// TIA Portal project "MOVIKIT_POSITIONING_V2.1_e_V15.1_V18" (V18)

(* hardware
DEVICE "S71500/ET200MP-Station_1"  S7-1500 station
   slot 0: "Profilschiene_0"  6ES7 590-1***0-0AA0
   slot 1: "S715xx"  CPU 1516F-3 PN/DP  6ES7 516-3FN00-0AB0  V1.8
DEVICE "SIMATIC 1200-Station_2"  S71200.Device
   slot 0: "S7-1200 Baugruppenträger"  Rack  V1.0
   slot 1: "S712xx"  CPU 1211C AC/DC/Rly  6ES7 211-1BD30-0XB0  V2.0
   slot 101: "CM 1243-5"  CM 1243-5  6GK7 243-5DX30-0XE0  V1.0
DEVICE "SIMATIC 300(1)"  S7-300 station
   slot 0: "Rack 0"  Rail  6ES7 390-1***0-0AA0
   slot 2: "CPU 315F-2 PN/DP"  CPU 315F-2 PN/DP  6ES7 315-2FH13-0AB0  V2.6
      slot 1: "MPI/DP interface_1"  X1
      slot 2: "PROFINET interface_1"  PN-IO
         slot 1: "Port_1"  Port
   slot 4: "DI 8/DO 8x24VDC/0.5A_1"  DI8/DO8 x 24VDC / 0.5A  6ES7 323-1BH01-0AA0
DEVICE "GSD-Geraet_1"  GSD.Device.PN
   slot 0: "Baugruppenträger"  Rack  V1.0
   slot 0: "pos-UDT-s73xx"  MDX90 + CFN21 V4.0
      slot 0: "MDX90 + CFN21 V4.0"  MDX90 + CFN21 V4.0
      slot 1: "PN-IO"  PN-IO
         slot 1: "Port 1 - RJ45 (X40)"  Port 1 - RJ45 (X40)
         slot 2: "Port 2 - RJ45 (X41)"  Port 2 - RJ45 (X41)
   slot 2: "Modul I/O (08 Worte)_1"  Module I/O (08 words)
      slot 0: "Modul I/O (08 Worte)"  Module I/O (08 words)
DEVICE "GSD-Geraet_2"  GSD.Device.PN
   slot 0: "Baugruppenträger"  Rack  V1.0
   slot 0: "pos-UDT-s712xx"  MDX90 + CFN21 V4.0
      slot 0: "MDX90 + CFN21 V4.0"  MDX90 + CFN21 V4.0
      slot 1: "PN-IO"  PN-IO
         slot 1: "Port 1 - RJ45 (X40)"  Port 1 - RJ45 (X40)
         slot 2: "Port 2 - RJ45 (X41)"  Port 2 - RJ45 (X41)
   slot 2: "Modul I/O (08 Worte)_1"  Module I/O (08 words)
      slot 0: "Modul I/O (08 Worte)"  Module I/O (08 words)
   slot 3: "Modul I/O (01 Wort)_1"  Module I/O (01 word)
      slot 0: "Modul I/O (01 Wort)"  Module I/O (01 word)
   slot 4: "Modul I/O (02 Worte)_1"  Module I/O (02 words)
      slot 0: "Modul I/O (02 Worte)"  Module I/O (02 words)
   slot 5: "Modul I/O (04 Worte)_1"  Module I/O (04 words)
      slot 0: "Modul I/O (04 Worte)"  Module I/O (04 words)
DEVICE "GSD-Geraet_4"  GSD.Device.PN
   slot 0: "Baugruppenträger"  Rack  V1.0
   slot 0: "pos-s712xx"  MDX90 + CFN21 V4.0
      slot 0: "MDX90 + CFN21 V4.0"  MDX90 + CFN21 V4.0
      slot 1: "PN-IO"  PN-IO
         slot 1: "Port 1 - RJ45 (X40)"  Port 1 - RJ45 (X40)
         slot 2: "Port 2 - RJ45 (X41)"  Port 2 - RJ45 (X41)
   slot 2: "Modul I/O (08 Worte)_1"  Module I/O (08 words)
      slot 0: "Modul I/O (08 Worte)"  Module I/O (08 words)
DEVICE "GSD-Geraet_3"  GSD.Device.PN
   slot 0: "Baugruppenträger"  Rack  V1.0
   slot 0: "pos-UDT-S715xx"  MDX90 + CFN21 V4.0
      slot 0: "MDX90 + CFN21 V4.0"  MDX90 + CFN21 V4.0
      slot 1: "PN-IO"  PN-IO
         slot 1: "Port 1 - RJ45 (X40)"  Port 1 - RJ45 (X40)
         slot 2: "Port 2 - RJ45 (X41)"  Port 2 - RJ45 (X41)
   slot 2: "Modul I/O (08 Worte)_1"  Module I/O (08 words)
      slot 0: "Modul I/O (08 Worte)"  Module I/O (08 words)
*)

// ===== PLC "S715xx"  CPU 1516F-3 PN/DP =====

VAR_GLOBAL   // PLC tag table "Standard-Variablentabelle"
   "Clock_Byte" AT %MB0 : Byte;
   "Clock_10Hz" AT %M0.0 : Bool;
   "Clock_5Hz" AT %M0.1 : Bool;
   "Clock_2.5Hz" AT %M0.2 : Bool;
   "Clock_2Hz" AT %M0.3 : Bool;
   "Clock_1.25Hz" AT %M0.4 : Bool;
   "Clock_1Hz" AT %M0.5 : Bool;
   "Clock_0.625Hz" AT %M0.6 : Bool;
   "Clock_0.5Hz" AT %M0.7 : Bool;
   "Reset" AT %M1000.0 : Bool;
   "set_ENABLE" AT %M1000.2 : Bool;
   "DRIVES_OFF" AT %M1000.1 : Bool;
   "POS_S715xx_Q" AT %A400.0 : "SEW_MOVIKIT_PositioningDrive_SETPOINTS_V2.1";   // Dieses UDT bildet die 5 Prozeßausgangsdaten der Funktion "Parameterkanal über Prozeßdaten" ab. This UDT maps the 5 process output data of the function "parameter channel via process data".
   "POS_S715xx_I" AT %E400.0 : "SEW_MOVIKIT_PositioningDrive_STATUS_V2.1";   // Dieses UDT bildet die 5 Prozeßeingangsdaten der Funktion "Parameterkanal über Prozeßdaten" ab. This UDT maps the 5 process input data of the function "parameter channel via process data"..
   "pos-plus-S715xx _Start" AT %M1001.7 : Bool;
   "Status (FCB)" AT %MW1004 : Int;
   "SubFault_Fault" AT %MW1024 : Word;
   "Fault" AT %MB1024 : SInt;
   "SubFault" AT %MB1025 : SInt;
   "pos-UDT-S715xx_PO1" AT %AW400 : Word;   // control word
   "pos-UDT-S715xx_PO2" AT %QW402 : Int;   // setpoint speed
   "pos-UDT-S715xx_PO3" AT %QW404 : Int;   // acceleration
   "pos-UDT-S715xx_PO4" AT %QW406 : Int;   // deceleration
   "pos-UDT-S715xx_PO5" AT %QW408 : Word;   // dig. Outputs
   "pos-UDT-S715xx_PI1" AT %IW400 : Int;   // status word
   "pos-UDT-S715xx_PI2" AT %IW402 : Int;   // actual speed
   "pos-UDT-S715xx_PI3" AT %IW404 : Word;   // Status/Main/Subfault
   "pos-UDT-S715xx_PI4" AT %IW406 : Int;   // actual torque
   "pos-UDT-S715xx_PI5" AT %IW408 : Word;   // dig. Inputs
   "pos-UDT-S715xx_PO6" AT %QW410 : Int;   // Target application mode
   "pos-UDT-S715xx_PO7-8" AT %QD412 : DInt;   // Target position
   "pos-UDT-S715xx_PI6" AT %IW416 : Int;   // actual application mode
   "pos-UDT-S715xx_PI7-8" AT %ID418 : DInt;   // actual position
END_VAR

TYPE "SEW_MOVIKIT_PositioningDrive_SETPOINTS_V2.1"
TITLE = SEW_MOVIKIT_PositioningDrive_SETPOINTS
// Dieses UDT bildet die 8 Prozeßeingangsdaten des MOVIKIT PositioningDrives ab. This UDT maps the 8 process input data of the MOVIKIT PositioningDrive.
   STRUCT
      x_Bit_8_Fault_Reset : Bool;
      x_Bit_9_Reserved : Bool;
      x_Bit_10_Activate_DriveTrain2 : Bool;
      x_Bit_11_Reserved : Bool;
      x_Bit_12_Deactivate_SW_Limit_switches : Bool;
      x_Bit_13_Activate_Output_Stage_Inhibit : Bool;
      x_Bit_14_Activate_StandBy_Mode : Bool;
      x_Bit_15_Heartbeat_IN : Bool;
      x_Bit_0_Enable_Emergency_Stop : Bool;
      x_Bit_1_Enable_Application_Stop : Bool;
      x_Bit_2_Reserved : Bool;
      x_Bit_3_Release_Brake : Bool;
      x_Bit_4_Jog_positive : Bool;
      x_Bit_5_Jog_negative : Bool;
      x_Bit_6_Apply_relative_Position : Bool;
      x_Bit_7_Start_Stop : Bool;
      iSetpoint_Speed : Int;
      iSetpoint_Acceleration : Int;
      iSetpoint_Deceleration : Int;
      wDigital_Outputs : Word;
      iSetpointApplicationMode : Int;
      diTargetPosition : DInt;
   END_STRUCT;
END_TYPE

TYPE "SEW_MOVIKIT_PositioningDrive_STATUS_V2.1"
TITLE = SEW_MOVIKIT_PositioningDrive_STATUS
// Dieses UDT bildet die 8 Prozeßausgangsdaten des MOVIKIT PositioningDrives ab. This UDT maps the 8 process output data of the MOVIKIT PositioningDrive.
   STRUCT
      x_Bit_8_Fault : Bool;
      x_Bit_9_Warning : Bool;
      x_Bit_10_DriveTrain2_active : Bool;
      x_Bit_11_Setp_actual_speed_comp_signal_active : Bool;
      x_Bit_12_SW_Limit_switches_inactive : Bool;
      x_Bit_13_Reserved : Bool;
      x_Bit_14_StandBy_mode_active : Bool;
      x_Bit_15_Heartbeat_OUT : Bool;
      x_Bit_0_Ready : Bool;
      x_Bit_1_STO_inactive : Bool;
      x_Bit_2_Output_Stage_enabled : Bool;
      x_Bit_3_Brake_released : Bool;
      x_Bit_4_Motor_turning : Bool;
      x_Bit_5_Active_Drive_referenced : Bool;
      x_Bit_6_New_Relative_Position_applied : Bool;
      x_Bit_7_In_Position_signal_active : Bool;
      iActual_Speed : Int;
      wStatus_main_fault_sub_fault : Word;
      iActual_Torque : Int;
      wDigital_Inputs : Word;
      iActual_Application_Mode : Int;
      diActual_Position : DInt;
   END_STRUCT;
END_TYPE

TYPE "SEW_MOVIKIT_5_PD_PAR_STATUS_V2.0"
   STRUCT
      x_Bit_8_READ_Service_selected : Bool;
      x_Bit_9_WRITE_Service_selected : Bool;
      x_Bit_10 : Bool;
      x_Bit_11 : Bool;
      x_Bit_12 : Bool;
      x_Bit_13_Service_active : Bool;
      x_Bit_14_Service_completed : Bool;
      x_Bit_15_Service_failed : Bool;
      x_Bit_0 : Bool;
      x_Bit_1 : Bool;
      x_Bit_2 : Bool;
      x_Bit_3 : Bool;
      x_Bit_4 : Bool;
      x_Bit_5 : Bool;
      x_Bit_6 : Bool;
      x_Bit_7 : Bool;
      i_actual_Index : Int;
      b_actual_SubIndex : Byte;
      b_actual_Offset : Byte;
      dw_value_read : DWord;
   END_STRUCT;
END_TYPE

TYPE "SEW_MOVIKIT_Function_torque_limit_STATUS_V2.0"
   STRUCT
      x_Bit_8 : Bool;
      x_Bit_9 : Bool;
      x_Bit_10 : Bool;
      x_Bit_11 : Bool;
      x_Bit_12 : Bool;
      x_Bit_13 : Bool;
      x_Bit_14 : Bool;
      x_Bit_15 : Bool;
      x_Bit_0_torque_limit_via_PD_active : Bool;
      x_Bit_1_speed_and_lag_error_monitoring_inactive : Bool;
      x_Bit_2_torque_limit_reached : Bool;
      x_Bit_3_speed_monitoring_inactive : Bool;
      x_Bit_4 : Bool;
      x_Bit_5 : Bool;
      x_Bit_6 : Bool;
      x_Bit_7 : Bool;
      i_actual_torque : Int;
   END_STRUCT;
END_TYPE

TYPE "SEW_MOVIKIT_5_PD_PAR_SETPOINTS_V2.0"
   STRUCT
      x_Bit_8_READ : Bool;
      x_Bit_9_WRITE : Bool;
      x_Bit_10 : Bool;
      x_Bit_11 : Bool;
      x_Bit_12 : Bool;
      x_Bit_13 : Bool;
      x_Bit_14_execute_function : Bool;
      x_Bit_15 : Bool;
      x_Bit_0 : Bool;
      x_Bit_1 : Bool;
      x_Bit_2 : Bool;
      x_Bit_3 : Bool;
      x_Bit_4 : Bool;
      x_Bit_5 : Bool;
      x_Bit_6 : Bool;
      x_Bit_7 : Bool;
      i_Index : Int;
      b_SubIndex : Byte;
      b_Offset : Byte;
      dw_value : DWord;
   END_STRUCT;
END_TYPE

TYPE "SEW_MOVIKIT_Function_torque_limit_SETPOINTS_V2.0"
   STRUCT
      x_Bit_8 : Bool;
      x_Bit_9 : Bool;
      x_Bit_10 : Bool;
      x_Bit_11 : Bool;
      x_Bit_12 : Bool;
      x_Bit_13 : Bool;
      x_Bit_14 : Bool;
      x_Bit_15 : Bool;
      x_Bit_0_activate_torque_limit_via_PD : Bool;
      x_Bit_1_deactivate_monitoring_of_speed_and_lag_error : Bool;
      x_Bit_2 : Bool;
      x_Bit_3_deactivate_speed_monitoring : Bool;
      x_Bit_4 : Bool;
      x_Bit_5 : Bool;
      x_Bit_6 : Bool;
      x_Bit_7 : Bool;
      i_maximum_torque : Int;
   END_STRUCT;
END_TYPE

TYPE "SEW_MOVIKIT_Function_touchprobe_STATUS_V2.0"
   STRUCT
      x_Bit_8 : Bool;
      x_Bit_9 : Bool;
      x_Bit_10 : Bool;
      x_Bit_11 : Bool;
      x_Bit_12 : Bool;
      x_Bit_13 : Bool;
      x_Bit_14 : Bool;
      x_Bit_15 : Bool;
      x_Bit_0_wait_for_trigger : Bool;
      x_Bit_1_trigger_activated : Bool;
      x_Bit_2_maximum_position_reached : Bool;
      x_Bit_3_touchprobe_travel_aborted : Bool;
      x_Bit_4 : Bool;
      x_Bit_5 : Bool;
      x_Bit_6 : Bool;
      x_Bit_7 : Bool;
      "i_counter_touchprobe 1" : Int;
      "di_detected_value_touchprobe 1" : DInt;
   END_STRUCT;
END_TYPE

TYPE "SEW_MOVIKIT_Function_touchprobe_SETPOINTS_V2.0"
   STRUCT
      x_Bit_8 : Bool;
      x_Bit_9 : Bool;
      x_Bit_10 : Bool;
      x_Bit_11 : Bool;
      x_Bit_12 : Bool;
      x_Bit_13 : Bool;
      x_Bit_14 : Bool;
      x_Bit_15 : Bool;
      x_Bit_0_activate_touchprobe_1 : Bool;
      x_Bit_1_activate_length_measurement : Bool;
      x_Bit_2 : Bool;
      x_Bit_3 : Bool;
      x_Bit_4 : Bool;
      x_Bit_5 : Bool;
      x_Bit_6 : Bool;
      x_Bit_7 : Bool;
      i_debouncing_time_for_length_measurement : Int;
      di_relative_position : DInt;
   END_STRUCT;
END_TYPE

FUNCTION "UDT_Positioning_Drive_example" : Void   // FC98, FBD
TITLE = Call the drive "pos-UDT-S715xx"
{ S7_Optimized_Access := 'TRUE' }
AUTHOR : SVSPASE
FAMILY : MOVIKIT
VERSION : 2.0
// This sample program only demonstrates the basic approach. We do not accept any legal or other liability for incorrect program functions and their consequences!
// 
// Please take note of the manual "MOVIKIT® Positioning, Velocity"
// 
// The UDTs "SEW_MOVIKIT_PositioningDrive_SETPOINTS_V2.1" and "SEW_MOVIKIT_PositioningDrive_STATUS_V2.1" are needed. Please make sure that the PLC data types are available in your TIA project.  These UDTs can be copied from the original TIA sample project or from the MOVIKIT_Vel_&_Pos_UDTs_V2.1.al14 library.
// 
// The plc tag "VELOCITY_S715xx_Q" has been assigned to the data type "SEW_MOVIKIT_PositioningDrive_SETPOINTS_V2.1" and  address Q400.0
// 
// The plc tag "VELOCITY_S715xx_I" has been assigned to the data type "SEW_MOVIKIT_PositioningDrive_STATUS_V2.1" and  address I400.0
BEGIN

REGION Network 1: Mapping of Status/Main fault/Subfault
   // If there is no fault or warning, the current FCB is output in "Status (FCB) MW1004 ).
   // 
   // If there is a fault or warning, the Subfault is copied in MB1024 and the Main fault in MB1025
   // 
   // => See "watch table "pos-UDT-S715xx"
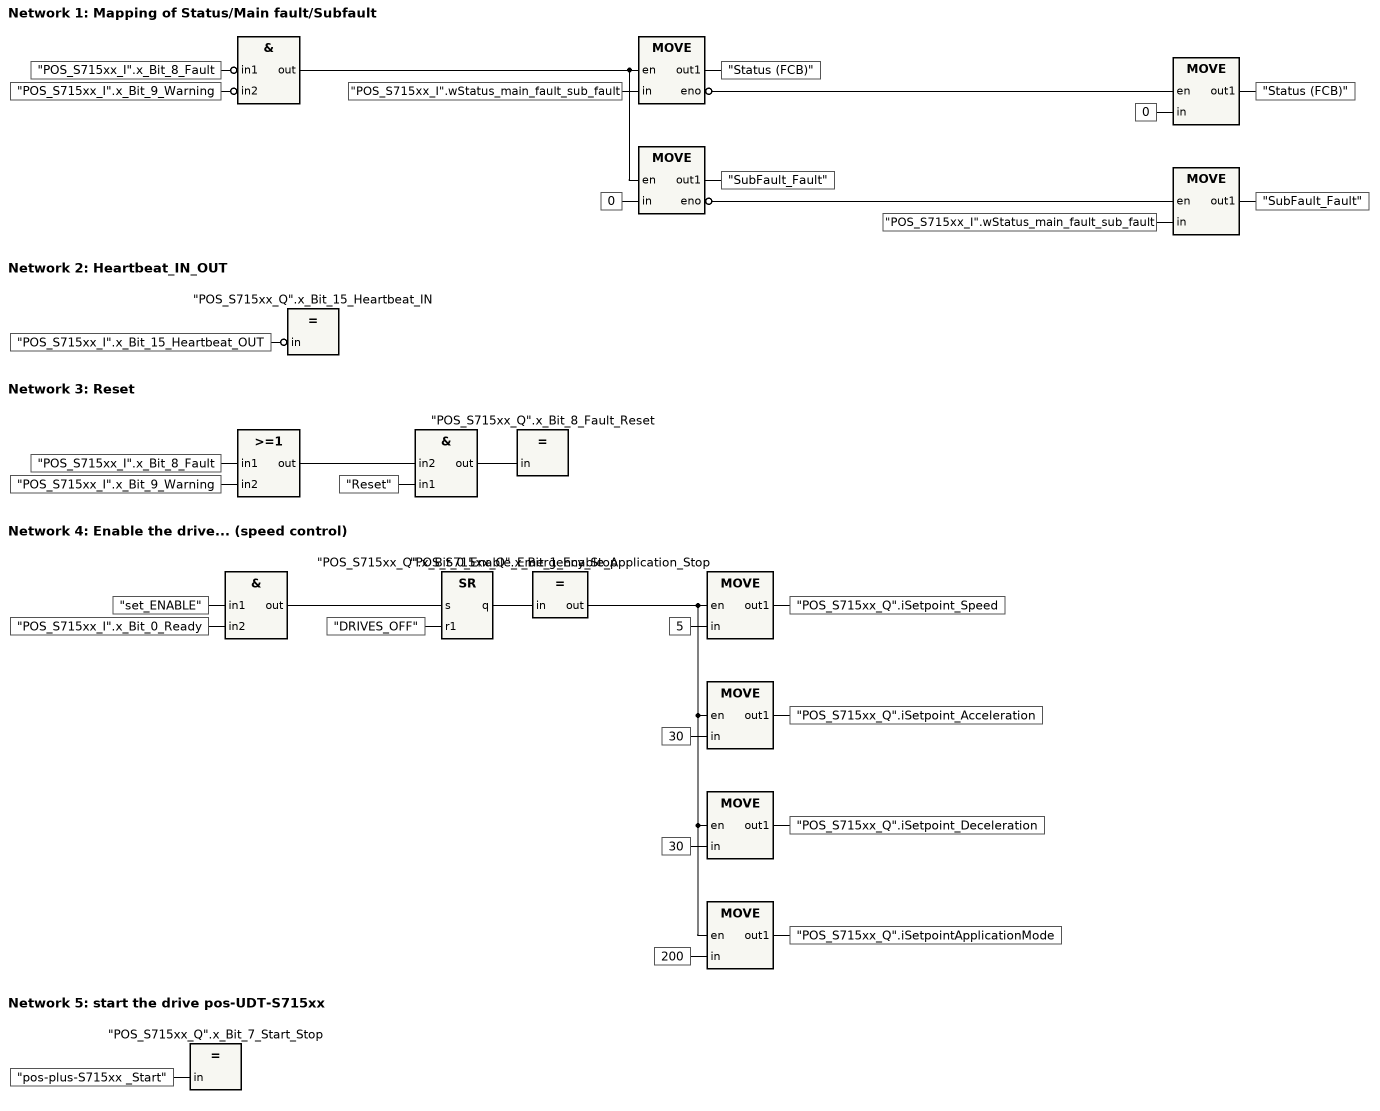
   IF NOT "POS_S715xx_I".x_Bit_8_Fault AND NOT "POS_S715xx_I".x_Bit_9_Warning THEN
       "Status (FCB)" := "POS_S715xx_I".wStatus_main_fault_sub_fault;
   END_IF;
   IF NOT (NOT "POS_S715xx_I".x_Bit_8_Fault AND NOT "POS_S715xx_I".x_Bit_9_Warning) THEN
       "Status (FCB)" := 0;
   END_IF;
   IF NOT "POS_S715xx_I".x_Bit_8_Fault AND NOT "POS_S715xx_I".x_Bit_9_Warning THEN
       "SubFault_Fault" := 0;
   END_IF;
   IF NOT (NOT "POS_S715xx_I".x_Bit_8_Fault AND NOT "POS_S715xx_I".x_Bit_9_Warning) THEN
       "SubFault_Fault" := "POS_S715xx_I".wStatus_main_fault_sub_fault;
   END_IF;
END_REGION

REGION Network 2: Heartbeat_IN_OUT
   "POS_S715xx_Q".x_Bit_15_Heartbeat_IN := NOT "POS_S715xx_I".x_Bit_15_Heartbeat_OUT;
END_REGION

REGION Network 3: Reset
   "POS_S715xx_Q".x_Bit_8_Fault_Reset := ("POS_S715xx_I".x_Bit_8_Fault OR "POS_S715xx_I".x_Bit_9_Warning) AND "Reset";
END_REGION

REGION Network 4: Enable the drive... (speed control)
   // - set enable
   // - assign setpoint speed, acceleration,..,.....
   IF "set_ENABLE" AND "POS_S715xx_I".x_Bit_0_Ready THEN
       "POS_S715xx_Q".x_Bit_0_Enable_Emergency_Stop := TRUE;   // SR flip-flop
   END_IF;
   IF "DRIVES_OFF" THEN "POS_S715xx_Q".x_Bit_0_Enable_Emergency_Stop := FALSE; END_IF;
   "POS_S715xx_Q".x_Bit_1_Enable_Application_Stop := "POS_S715xx_Q".x_Bit_0_Enable_Emergency_Stop;
   IF "POS_S715xx_Q".x_Bit_0_Enable_Emergency_Stop THEN
       "POS_S715xx_Q".iSetpoint_Speed := 5;
       "POS_S715xx_Q".iSetpoint_Acceleration := 30;
       "POS_S715xx_Q".iSetpoint_Deceleration := 30;
       "POS_S715xx_Q".iSetpointApplicationMode := 200;
   END_IF;
END_REGION

REGION Network 5: start the drive pos-UDT-S715xx
   "POS_S715xx_Q".x_Bit_7_Start_Stop := "pos-plus-S715xx _Start";
END_REGION
END_FUNCTION

ORGANIZATION_BLOCK "Main"   // OB1, STL, ProgramCycle
TITLE = "Main Program Sweep (Cycle)"
{ S7_Optimized_Access := 'FALSE' }
VERSION : 0.1
// This sample program only demonstrates the basic approach. We do not accept any legal or other liability for incorrect program functions and their consequences!
// 
// Please take note of the manual "MOVIKIT® Positioning, Velocity"
   VAR_TEMP
      OB1_EV_CLASS : Byte;   // Bits 0-3 = 1 (Coming event), Bits 4-7 = 1 (Event class 1)
      OB1_SCAN_1 : Byte;   // 1 (Cold restart scan 1 of OB 1), 3 (Scan 2-n of OB 1)
      OB1_PRIORITY : Byte;   // Priority of OB Execution
      OB1_OB_NUMBR : Byte;   // 1 (Organization block 1, OB1)
      OB1_RESERVED_1 : Byte;   // Reserved for system
      OB1_RESERVED_2 : Byte;   // Reserved for system
      OB1_PREV_CYCLE : Int;   // Cycle time of previous OB1 scan (milliseconds)
      OB1_MIN_CYCLE : Int;   // Minimum cycle time of OB1 (milliseconds)
      OB1_MAX_CYCLE : Int;   // Maximum cycle time of OB1 (milliseconds)
      OB1_DATE_TIME : Date_And_Time;   // Date and time OB1 started
   END_VAR
BEGIN

REGION Network 1: Call the drive "velocity-UDT-S715xx"

         CALL  "UDT_Positioning_Drive_example";
END_REGION
END_ORGANIZATION_BLOCK

// ===== PLC "S712xx"  CPU 1211C AC/DC/Rly =====

VAR_GLOBAL   // PLC tag table "Standard-Variablentabelle"
   "Clock_Byte" AT %MB0 : Byte;
   "Clock_10Hz" AT %M0.0 : Bool;
   "Clock_5Hz" AT %M0.1 : Bool;
   "Clock_2.5Hz" AT %M0.2 : Bool;
   "Clock_2Hz" AT %M0.3 : Bool;
   "Clock_1.25Hz" AT %M0.4 : Bool;
   "Clock_1Hz" AT %M0.5 : Bool;
   "Clock_0.625Hz" AT %M0.6 : Bool;
   "Clock_0.5Hz" AT %M0.7 : Bool;
   "pos-UDT-S712xx_PO9_Jerk_Time" AT %QW316 : Int;   // Slot 3: jerk time
   "pos-S712xx_PO1" AT %QW330 : Int;   // control word
   "pos-S712xx_PO2" AT %QW332 : Int;   // setpoint speed
   "pos-S712xx_PO3" AT %QW334 : Int;   // acceleration
   "pos-S712xx_PO4" AT %QW336 : Int;   // deceleration
   "pos-S712xx_PO5" AT %QW338 : Int;   // dig. Outputs
   "pos-S712xx_PI1" AT %IW330 : Int;   // status word
   "pos-S712xx_PI2" AT %IW332 : Int;   // actual speed
   "pos-S712xx_PI3" AT %IW334 : Int;   // Status/Main/Subfault
   "pos-S712xx_PI4" AT %IW336 : Int;   // actual torque
   "pos-S712xx_PI5" AT %IW338 : Int;   // dig. Inputs
   "pos-UDT-S712xx_PO1" AT %QW300 : Int;   // Slot 2: control word
   "pos-UDT-S712xx_PO2" AT %QW302 : Int;   // Slot 2: setpoint speed
   "pos-UDT-S712xx_PO3" AT %QW304 : Int;   // Slot 2: acceleration
   "pos-UDT-S712xx_PO4" AT %QW306 : Int;   // Slot 2: deceleration
   "pos-UDT-S712xx_PO5" AT %QW308 : Word;   // Slot 2: dig. Outputs
   "pos-UDT-S712xx_PI1" AT %IW300 : Word;   // Slot 2: status word
   "pos-UDT-S712xx_PI2" AT %IW302 : Int;   // Slot 2: actual speed
   "pos-UDT-S712xx_PI3" AT %IW304 : Int;   // Slot 2: Status/Main/Subfault
   "pos-UDT-S712xx_PI4" AT %IW306 : Int;   // Slot 2: actual torque
   "pos-UDT-S712xx_PI5" AT %IW308 : Int;   // Slot 2: dig. Inputs
   "pos-UDT-S712xx_PI6" AT %IW310 : Int;   // Slot 2: actual application mode
   "pos-UDT-S712xx_PI7-8" AT %ID312 : DInt;   // Slot 2: actual position
   "pos-UDT-S712xx_PI9" AT %IW316 : Int;   // Slot 3: reserved
   "pos-UDT-S712xx_PI10" AT %IW318 : Int;   // Slot 4: Status word for torque limit
   "pos-UDT-S712xx_PI11" AT %IW320 : Int;   // Slot 4: Acual torque
   "pos-UDT-S712xx_PI12" AT %IW322 : Word;   // Slot 5: Status word for positioning via touchprobe
   "pos-S712xx_PO6" AT %QW340 : Int;   // target application mode
   "pos-S712xx_PO7-8" AT %QD342 : DInt;   // target position
   "pos-S712xx_PI6" AT %IW340 : Int;   // actual application mode
   "pos-S712xx_PI7-8" AT %ID342 : DInt;   // actual position
   "pos-UDT-S712xx_PO6" AT %QW310 : Int;   // Slot 2: target application mode
   "pos-UDT-S712xx_PO7-8" AT %QD312 : DInt;   // Slot 2: Target position
   "pos-UDT-S712xx_PO10" AT %QW318 : Word;   // Slot 4: Control word for torque limit
   "pos-UDT-S712xx_PO11" AT %QW320 : Int;   // Slot 4: Maximum Torque
   "pos-UDT-S712xx_PO12" AT %QW322 : Word;   // Slot 5: Control word for pos. via touch probe
   "pos-UDT-S712xx_PO13" AT %QW324 : Int;   // Slot 5: Debouncing time for length measurement
   "pos-UDT-S712xx_PO14-15" AT %QD326 : DInt;   // Slot 5: relative position
   "pos-UDT-S712xx_PI13" AT %IW324 : Int;   // Slot 5: Counter Touch probe 1
   "pos-UDT-S712xx_PI4-15" AT %ID326 : DInt;   // Slot 5: detected value touchprobe 1
END_VAR

TYPE "SEW_MOVIKIT_PositioningDrive_SETPOINTS_V2.1"
TITLE = SEW_MOVIKIT_PositioningDrive_SETPOINTS
// Dieses UDT bildet die 8 Prozeßeingangsdaten des MOVIKIT PositioningDrives ab. This UDT maps the 8 process input data of the MOVIKIT PositioningDrive.
   STRUCT
      x_Bit_8_Fault_Reset : Bool;
      x_Bit_9_Reserved : Bool;
      x_Bit_10_Activate_DriveTrain2 : Bool;
      x_Bit_11_Reserved : Bool;
      x_Bit_12_Deactivate_SW_Limit_switches : Bool;
      x_Bit_13_Activate_Output_Stage_Inhibit : Bool;
      x_Bit_14_Activate_StandBy_Mode : Bool;
      x_Bit_15_Heartbeat_IN : Bool;
      x_Bit_0_Enable_Emergency_Stop : Bool;
      x_Bit_1_Enable_Application_Stop : Bool;
      x_Bit_2_Reserved : Bool;
      x_Bit_3_Release_Brake : Bool;
      x_Bit_4_Jog_positive : Bool;
      x_Bit_5_Jog_negative : Bool;
      x_Bit_6_Apply_relative_Position : Bool;
      x_Bit_7_Start_Stop : Bool;
      iSetpoint_Speed : Int;
      iSetpoint_Acceleration : Int;
      iSetpoint_Deceleration : Int;
      wDigital_Outputs : Word;
      iSetpointApplicationMode : Int;
      diTargetPosition : DInt;
   END_STRUCT;
END_TYPE

TYPE "SEW_MOVIKIT_PositioningDrive_STATUS_V2.1"
TITLE = SEW_MOVIKIT_PositioningDrive_STATUS
// Dieses UDT bildet die 8 Prozeßausgangsdaten des MOVIKIT PositioningDrives ab. This UDT maps the 8 process output data of the MOVIKIT PositioningDrive.
   STRUCT
      x_Bit_8_Fault : Bool;
      x_Bit_9_Warning : Bool;
      x_Bit_10_DriveTrain2_active : Bool;
      x_Bit_11_Setp_actual_speed_comp_signal_active : Bool;
      x_Bit_12_SW_Limit_switches_inactive : Bool;
      x_Bit_13_Reserved : Bool;
      x_Bit_14_StandBy_mode_active : Bool;
      x_Bit_15_Heartbeat_OUT : Bool;
      x_Bit_0_Ready : Bool;
      x_Bit_1_STO_inactive : Bool;
      x_Bit_2_Output_Stage_enabled : Bool;
      x_Bit_3_Brake_released : Bool;
      x_Bit_4_Motor_turning : Bool;
      x_Bit_5_Active_Drive_referenced : Bool;
      x_Bit_6_New_Relative_Position_applied : Bool;
      x_Bit_7_In_Position_signal_active : Bool;
      iActual_Speed : Int;
      wStatus_main_fault_sub_fault : Word;
      iActual_Torque : Int;
      wDigital_Inputs : Word;
      iActual_Application_Mode : Int;
      diActual_Position : DInt;
   END_STRUCT;
END_TYPE

TYPE "SEW_MOVIKIT_5_PD_PAR_STATUS_V2.0"
   STRUCT
      x_Bit_8_READ_Service_selected : Bool;
      x_Bit_9_WRITE_Service_selected : Bool;
      x_Bit_10 : Bool;
      x_Bit_11 : Bool;
      x_Bit_12 : Bool;
      x_Bit_13_Service_active : Bool;
      x_Bit_14_Service_completed : Bool;
      x_Bit_15_Service_failed : Bool;
      x_Bit_0 : Bool;
      x_Bit_1 : Bool;
      x_Bit_2 : Bool;
      x_Bit_3 : Bool;
      x_Bit_4 : Bool;
      x_Bit_5 : Bool;
      x_Bit_6 : Bool;
      x_Bit_7 : Bool;
      i_actual_Index : Int;
      b_actual_SubIndex : Byte;
      b_actual_Offset : Byte;
      dw_value_read : DWord;
   END_STRUCT;
END_TYPE

TYPE "SEW_MOVIKIT_Function_torque_limit_STATUS_V2.0"
   STRUCT
      x_Bit_8 : Bool;
      x_Bit_9 : Bool;
      x_Bit_10 : Bool;
      x_Bit_11 : Bool;
      x_Bit_12 : Bool;
      x_Bit_13 : Bool;
      x_Bit_14 : Bool;
      x_Bit_15 : Bool;
      x_Bit_0_torque_limit_via_PD_active : Bool;
      x_Bit_1_speed_and_lag_error_monitoring_inactive : Bool;
      x_Bit_2_torque_limit_reached : Bool;
      x_Bit_3_speed_monitoring_inactive : Bool;
      x_Bit_4 : Bool;
      x_Bit_5 : Bool;
      x_Bit_6 : Bool;
      x_Bit_7 : Bool;
      i_actual_torque : Int;
   END_STRUCT;
END_TYPE

TYPE "SEW_MOVIKIT_5_PD_PAR_SETPOINTS_V2.0"
   STRUCT
      x_Bit_8_READ : Bool;
      x_Bit_9_WRITE : Bool;
      x_Bit_10 : Bool;
      x_Bit_11 : Bool;
      x_Bit_12 : Bool;
      x_Bit_13 : Bool;
      x_Bit_14_execute_function : Bool;
      x_Bit_15 : Bool;
      x_Bit_0 : Bool;
      x_Bit_1 : Bool;
      x_Bit_2 : Bool;
      x_Bit_3 : Bool;
      x_Bit_4 : Bool;
      x_Bit_5 : Bool;
      x_Bit_6 : Bool;
      x_Bit_7 : Bool;
      i_Index : Int;
      b_SubIndex : Byte;
      b_Offset : Byte;
      dw_value : DWord;
   END_STRUCT;
END_TYPE

TYPE "SEW_MOVIKIT_Function_torque_limit_SETPOINTS_V2.0"
   STRUCT
      x_Bit_8 : Bool;
      x_Bit_9 : Bool;
      x_Bit_10 : Bool;
      x_Bit_11 : Bool;
      x_Bit_12 : Bool;
      x_Bit_13 : Bool;
      x_Bit_14 : Bool;
      x_Bit_15 : Bool;
      x_Bit_0_activate_torque_limit_via_PD : Bool;
      x_Bit_1_deactivate_monitoring_of_speed_and_lag_error : Bool;
      x_Bit_2 : Bool;
      x_Bit_3_deactivate_speed_monitoring : Bool;
      x_Bit_4 : Bool;
      x_Bit_5 : Bool;
      x_Bit_6 : Bool;
      x_Bit_7 : Bool;
      i_maximum_torque : Int;
   END_STRUCT;
END_TYPE

TYPE "SEW_MOVIKIT_Function_touchprobe_STATUS_V2.0"
   STRUCT
      x_Bit_8 : Bool;
      x_Bit_9 : Bool;
      x_Bit_10 : Bool;
      x_Bit_11 : Bool;
      x_Bit_12 : Bool;
      x_Bit_13 : Bool;
      x_Bit_14 : Bool;
      x_Bit_15 : Bool;
      x_Bit_0_wait_for_trigger : Bool;
      x_Bit_1_trigger_activated : Bool;
      x_Bit_2_maximum_position_reached : Bool;
      x_Bit_3_touchprobe_travel_aborted : Bool;
      x_Bit_4 : Bool;
      x_Bit_5 : Bool;
      x_Bit_6 : Bool;
      x_Bit_7 : Bool;
      "i_counter_touchprobe 1" : Int;
      "di_detected_value_touchprobe 1" : DInt;
   END_STRUCT;
END_TYPE

TYPE "SEW_MOVIKIT_Function_touchprobe_SETPOINTS_V2.0"
   STRUCT
      x_Bit_8 : Bool;
      x_Bit_9 : Bool;
      x_Bit_10 : Bool;
      x_Bit_11 : Bool;
      x_Bit_12 : Bool;
      x_Bit_13 : Bool;
      x_Bit_14 : Bool;
      x_Bit_15 : Bool;
      x_Bit_0_activate_touchprobe_1 : Bool;
      x_Bit_1_activate_length_measurement : Bool;
      x_Bit_2 : Bool;
      x_Bit_3 : Bool;
      x_Bit_4 : Bool;
      x_Bit_5 : Bool;
      x_Bit_6 : Bool;
      x_Bit_7 : Bool;
      i_debouncing_time_for_length_measurement : Int;
      di_relative_position : DInt;
   END_STRUCT;
END_TYPE

DATA_BLOCK "Pos_269"   // DB269
{ S7_Optimized_Access := 'FALSE' }
VERSION : 0.1
   VAR
      PO : "SEW_MOVIKIT_PositioningDrive_SETPOINTS_V2.1";
      PI : "SEW_MOVIKIT_PositioningDrive_STATUS_V2.1";
      Communication_OK : Bool;   // true: DPRD_DAT u. DPWR_DAT arbeiten fehlerfrei. false: 5-PD-Steckplatz erforderlich; Adresse an Eingang "IO_ADDRESS" überprüfen
   END_VAR
BEGIN
END_DATA_BLOCK

DATA_BLOCK "TORQUE_278"   // DB278
{ S7_Optimized_Access := 'FALSE' }
VERSION : 0.1
   VAR
      HW_IDENTIFIER : Hw_Io := 278;
      ACTIVATE_TORQUE_LIMIT_VIA_PD : Bool;
      DEACTIVATE_MONITORING_OF_SPEED_LAG_ERROR : Bool;
      DEACTIVATE_SPEED_MONITORING : Bool;
      MAXIMUM_TORQUE : Int;
      COMMUNICATION_OK : Bool;
      TORQUE_LIMIT_VIA_PD_ACTIVE : Bool;
      SPEED_LAG_ERROR_MONITORING_INACTIVE : Bool;
      TORQUE_LIMIT_REACHED : Bool;
      SPEED_MONITORING_INACTIVE : Bool;
      ACTUAL_TORQUE : Int;
   END_VAR
BEGIN
END_DATA_BLOCK

DATA_BLOCK "TOUCHPROBE_279"   // DB279
{ S7_Optimized_Access := 'FALSE' }
VERSION : 0.1
   VAR
      PO : "SEW_MOVIKIT_Function_touchprobe_SETPOINTS_V2.0";
      PI : "SEW_MOVIKIT_Function_touchprobe_STATUS_V2.0";
      Communication_OK : Bool;
   END_VAR
BEGIN
END_DATA_BLOCK

DATA_BLOCK "Pos_291"   // DB291
{ S7_Optimized_Access := 'FALSE' }
VERSION : 0.1
   VAR
      ENABLE_EMERGENCY_STOP : Bool;
      ENABLE_APPLICATION_STOP : Bool;
      RELEASE_BRAKE : Bool;
      JOG_POSITIVE : Bool;   // true: Jog positive
      JOG_NEGATIVE : Bool;   // true: Jog negative
      APPLY_RELATIVE_POSITION : Bool;   // true: Apply relative position
      START_STOP : Bool;
      FAULT_RESET : Bool;
      ACTIVATE_DRIVE_TRAIN_2 : Bool;
      DEACTIVATE_SW_LIMIT_SWITCH : Bool;
      ACTIVATE_OUTPUT_STAGE_INHIBIT : Bool;
      ACTIVATE_STANDBY_MODE : Bool;
      HEARTBEAT_IN : Bool;
      SETPOINT_SPEED : Int;
      SETPOINT_ACCELERATION : Int;
      SETPOINT_DECELERATION : Int;
      DIGITAL_OUTPUTS : Word;
      SETPOINT_APPLICATION_MODE : Int;   // Operating_Mode: 10x: Jog; 30x: Ref.; 40x: Pos.; 700: Brake test => Manual "MOVIKIT® Positioning, Velocity"
      TARGET_POSITION : DInt;   // Target Position in user unit
      COMMUNICATION_OK : Bool;
      READY : Bool;
      STO_INACTIVE : Bool;
      OUTPUT_STAGE_ENABLED : Bool;
      BRAKE_RELEASED : Bool;
      MOTOR_TURNING : Bool;
      ACTIVE_DRIVE_REFERENCED : Bool;   // true: Active drive referenced
      NEW_RELATIVE_POSITION_APPLIED : Bool;   // true: New relative position applied
      IN_POSITION_SIGNAL_ACTIVE : Bool;
      FAULT : Bool;
      WARNING : Bool;
      DRIVE_TRAIN_2_ACTIVE : Bool;
      SETP_ACTUAL_SPEED_COMPARISON_SIGNAL_ACTIVE : Bool;
      SW_LIMIT_SWITCH_INACTIVE : Bool;
      STANDBY_MODE_ACTIVE : Bool;
      HEARTBEAT_OUT : Bool;
      ACTUAL_SPEED : Int;
      STATUS_MAIN_FAULT_SUB_FAULT : Int;
      ACTUAL_TORQUE : Int;
      DIGITAL_INPUTS : Word;
      ACTUAL_APPLICATION_MODE : Int;   // Actual Operating_Mode: 10x: Jog; 30x: Ref.; 40x: Pos.; 700: Brake test => Manual "MOVIKIT® Positioning, Velocity"
      ACTUAL_POSITION : DInt;   // Actual Position in user unit
   END_VAR
BEGIN
END_DATA_BLOCK

FUNCTION "Call pos-S712xx" : Void   // FC100, FBD
TITLE = Call pos-S712xx
{ S7_Optimized_Access := 'TRUE' }
VERSION : 0.1
// This sample program only demonstrates the basic approach. We do not accept any legal or other liability for incorrect program functions and their consequences!
// 
// Please take note of the manual "MOVIKIT® Positioning, Velocity"
BEGIN

REGION Network 1: Call pos-S712xx
   // The FC140 serves as a program module for controlling the MOVIKIT module "Positioning Drive" for the Generation C device series. With the help of the FC140, the converters can be controlled via PROFINET IO/PROFIBUS DP. 
   // 
   // Device & networks: To use this FC, a 8 PD slot must be configured.
   // 
   // Inputs of the FC:
   // 
   // "IO_ADDRESS": Assign the HW-Identifier of the 8 PD slot. 
   // 
   // "ENABLE_EMERGENCY_STOP" = true: Enable; false: emergency stop
   // "ENABLE_APPLICATION_STOP" = true: Enable; false: Application stop
   // "RELEASE_BRAKE" = true: release brake (without enable)
   // "JOG_POSITIVE": Signal for moving the drive in positive direction in jog mode.
   // "JOG_NEGATIVE": Signal for moving the drive in negative direction in jog mode.
   // "Apply relative position": Apply relative target position in relative positioning mode (401).
   // "START_STOP" = Start/stop with fieldbus ramp
   // "FAULT_RESET": true: Fault reset
   // "ACTIVATE_DRIVE_TRAIN_2" = true: Activate drive train 2
   // "DEACTIVATE_SW_LIMIT_SWITCH"
   // "ACTIVATE_OUPUT_STAGE_INHIBIT" = true: Activate output stage inhibit
   // "ACTIVATE_STANDBY_MODE" = true: Activate standby mode
   // "HEARTBEAT_IN": Copied to HEARTBEAT_OUT
   // "SETPOINT_SPEED": in user unit (INT) 
   // "SETPOINT_ACCELERATION":  in user unit (INT) 
   // "SETPOINT_DECELERATION":  in user unit (INT)
   // "DIGITAL_OUTPUTS": MoviSuite/Movikit../Inputs/Outputs: dig Outputs: the setting "control via fieldbus" is needed
   // "SETPOINT_APPLICATION_MODE": Operating_Mode: 10x: Jog; 30x: Ref.; 40x: Pos.; 700: Brake test 
   //     => Manual "MOVIKIT® Positioning, Velocity"
   // "TARGET_POSITION":	Target Position in user unit (DINT)
   // 
   // Outputs of the FC:
   // 
   // If the data transmission/PROFINET is disrupted, all outputs will be deleted..
   // => "COMMUNICATION_OK = false (self-confirming)
   // "READY" = true: Ready for operation.
   // "STO_INACTIVE" = true: STO inactive.
   // "OUTPUT_STAGE_ENABLED" = true: Output stage enabled.
   // "BRAKE_RELEASED" = true: Brake released.
   // "MOTOR_TURNING" = true: Motor running
   // "ACTIVE_DRIVE_REFERENCED" = true: Active drive referenced
   // "NEW_RELATIVE_POSITION_APPLIED" = true: New relative position applied
   // "IN_POSITION_SIGNAL_ACTIVE" = true: "In position" signal active
   // "FAULT" = true: Fault.
   // "WARNING" = true: Warning 
   // "DRIVE_TRAIN_2_ACTIVE" = true: Drive train 2 active.
   // "SETPOINT-ACTUAL_COMPARISON"
   // "SW_LIMIT_SWITCHES_INACTIVE" = true: Software limit switches inactive
   //  "STANDBY_MODE_INACTIVE" = true: Stand-by Mode is active.
   // "HEARTBEAT_OUT" : This signal is copied internally from "HEARTBEAT_IN"
   // "ACTUAL_SPEED": in user unit (INT) 
   // "STATUS_MAIN_FAULT_SUB_FAULT:" (WORD)
   //    No fault: Display of current FCB; fault/warning:  High-Byte Fault; Low-Byte SubFault
   // "ACTUAL_TORQUE":in user unit (INT)
   // "DIGITAL_INPUTS" : The digital inputs are read out
   // "ACTUAL_APPLICATION_MODE":	Actual Operating_Mode: 10x: Jog; 30x: Ref.; 40x: Pos.; 700: Brake test 
   //     => Manual "MOVIKIT® Positioning, Velocity"
   // "ACTUAL_POSITION":	 Actual Position in user unit (DINT)
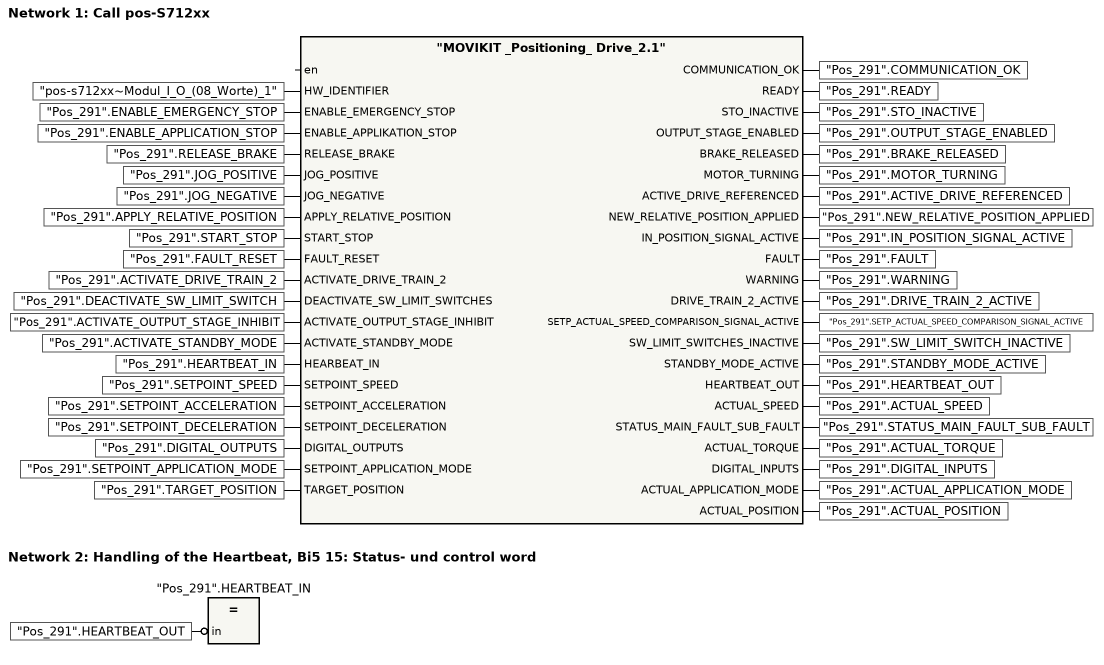
   "MOVIKIT _Positioning_ Drive_2.1"(HW_IDENTIFIER := "pos-s712xx~Modul_I_O_(08_Worte)_1",
                           ENABLE_EMERGENCY_STOP := "Pos_291".ENABLE_EMERGENCY_STOP,
                           ENABLE_APPLIKATION_STOP := "Pos_291".ENABLE_APPLICATION_STOP,
                           RELEASE_BRAKE := "Pos_291".RELEASE_BRAKE,
                           JOG_POSITIVE := "Pos_291".JOG_POSITIVE,
                           JOG_NEGATIVE := "Pos_291".JOG_NEGATIVE,
                           APPLY_RELATIVE_POSITION := "Pos_291".APPLY_RELATIVE_POSITION,
                           START_STOP := "Pos_291".START_STOP,
                           FAULT_RESET := "Pos_291".FAULT_RESET,
                           ACTIVATE_DRIVE_TRAIN_2 := "Pos_291".ACTIVATE_DRIVE_TRAIN_2,
                           DEACTIVATE_SW_LIMIT_SWITCHES := "Pos_291".DEACTIVATE_SW_LIMIT_SWITCH,
                           ACTIVATE_OUTPUT_STAGE_INHIBIT := "Pos_291".ACTIVATE_OUTPUT_STAGE_INHIBIT,
                           ACTIVATE_STANDBY_MODE := "Pos_291".ACTIVATE_STANDBY_MODE,
                           HEARBEAT_IN := "Pos_291".HEARTBEAT_IN,
                           SETPOINT_SPEED := "Pos_291".SETPOINT_SPEED,
                           SETPOINT_ACCELERATION := "Pos_291".SETPOINT_ACCELERATION,
                           SETPOINT_DECELERATION := "Pos_291".SETPOINT_DECELERATION,
                           DIGITAL_OUTPUTS := "Pos_291".DIGITAL_OUTPUTS,
                           SETPOINT_APPLICATION_MODE := "Pos_291".SETPOINT_APPLICATION_MODE,
                           TARGET_POSITION := "Pos_291".TARGET_POSITION,
                           COMMUNICATION_OK => "Pos_291".COMMUNICATION_OK,
                           READY => "Pos_291".READY,
                           STO_INACTIVE => "Pos_291".STO_INACTIVE,
                           OUTPUT_STAGE_ENABLED => "Pos_291".OUTPUT_STAGE_ENABLED,
                           BRAKE_RELEASED => "Pos_291".BRAKE_RELEASED,
                           MOTOR_TURNING => "Pos_291".MOTOR_TURNING,
                           ACTIVE_DRIVE_REFERENCED => "Pos_291".ACTIVE_DRIVE_REFERENCED,
                           NEW_RELATIVE_POSITION_APPLIED => "Pos_291".NEW_RELATIVE_POSITION_APPLIED,
                           IN_POSITION_SIGNAL_ACTIVE => "Pos_291".IN_POSITION_SIGNAL_ACTIVE,
                           FAULT => "Pos_291".FAULT,
                           WARNING => "Pos_291".WARNING,
                           DRIVE_TRAIN_2_ACTIVE => "Pos_291".DRIVE_TRAIN_2_ACTIVE,
                           SETP_ACTUAL_SPEED_COMPARISON_SIGNAL_ACTIVE => "Pos_291".SETP_ACTUAL_SPEED_COMPARISON_SIGNAL_ACTIVE,
                           SW_LIMIT_SWITCHES_INACTIVE => "Pos_291".SW_LIMIT_SWITCH_INACTIVE,
                           STANDBY_MODE_ACTIVE => "Pos_291".STANDBY_MODE_ACTIVE,
                           HEARTBEAT_OUT => "Pos_291".HEARTBEAT_OUT,
                           ACTUAL_SPEED => "Pos_291".ACTUAL_SPEED,
                           STATUS_MAIN_FAULT_SUB_FAULT => "Pos_291".STATUS_MAIN_FAULT_SUB_FAULT,
                           ACTUAL_TORQUE => "Pos_291".ACTUAL_TORQUE,
                           DIGITAL_INPUTS => "Pos_291".DIGITAL_INPUTS,
                           ACTUAL_APPLICATION_MODE => "Pos_291".ACTUAL_APPLICATION_MODE,
                           ACTUAL_POSITION => "Pos_291".ACTUAL_POSITION);
END_REGION

REGION Network 2: Handling of the Heartbeat, Bi5 15: Status- und control word
   "Pos_291".HEARTBEAT_IN := NOT "Pos_291".HEARTBEAT_OUT;
END_REGION
END_FUNCTION

FUNCTION "Call_pos-UDT-S712xx" : Void   // FC101, FBD
TITLE = Control of the drive pos-UDT-S712xx with the functions "Variable jerk time, Variable torque limitation, touchprobe
{ S7_Optimized_Access := 'TRUE' }
VERSION : 0.1
// This sample program only demonstrates the basic approach. We do not accept any legal or other liability for incorrect program functions and their consequences!
// 
// Please take note of the manual "MOVIKIT® Positioning, Velocity"
// 
// Control of the MOVIKITS Velocity Drive with the functions "Variable jerk time, Variable torque limitation,  touchprobe.
BEGIN

REGION Network 1: Slot 2, PD 1..8: Control of the drive pos-UDT-S712xx
   // The FC141 serves as a program module for controlling the MOVIKIT module "Positioning Drive" for the Generation C device series. With the help of the FC141, the converters can be controlled via PROFINET IO/PROFIBUS DP. 
   // 
   // Device & networks: To use this FC, a 8 PD slot must be configured.
   // 
   // This FC uses the UDTs "SEW_MOVIKIT_PositioningDrive_SETPOINTS_V2.1" and "SEW_MOVIKIT_PositioningDrive_STATUS_V2.1". Please make sure that these PLC data types are available in your TIA project. These UDTs can be copied from the original TIA sample project or from the MOVIKIT_POSITIONING_UDTs_V2.x.al14 library.
   // 
   // Inputs of the FC:
   // 
   // Attention! 
   // S71xxx: "HW_Identifier". Assign the HW-Identifier of the 8 PD slot. 
   // S73xx/4xx:"HW_Identifier"Change the data type from "HW_IO" to "WORD" Assign the peripheral address of the 8 PD slot;
   // 
   // "ENABLE_EMERGENCY_STOP" = true: Enable; false: emergency stop
   // "ENABLE_APPLICATION_STOP" = true: Enable; false: Application stop
   // "RELEASE_BRAKE" = true: release brake (without enable)
   // "JOG_POSITIVE": Signal for moving the drive in positive direction in jog mode.
   // "JOG_NEGATIVE": Signal for moving the drive in negative direction in jog mode.
   // "Apply relative position": Apply relative target position in relative positioning mode (401).
   // "START_STOP" = Start/stop with fieldbus ramp
   // "FAULT_RESET": true: Fault reset
   // "ACTIVATE_DRIVE_TRAIN_2" = true: Activate drive train 2
   // "DEACTIVATE_SW_LIMIT_SWITCH"
   // "ACTIVATE_OUPUT_STAGE_INHIBIT" = true: Activate output stage inhibit
   // "ACTIVATE_STANDBY_MODE" = true: Activate standby mode
   // "HEARTBEAT_IN": Copied to HEARTBEAT_OUT
   // "SETPOINT_SPEED": in user unit (INT) 
   // "SETPOINT_ACCELERATION":  in user unit (INT) 
   // "SETPOINT_DECELERATION":  in user unit (INT)
   // "DIGITAL_OUTPUTS": MoviSuite/Movikit../Inputs/Outputs: dig Outputs: the setting "control via fieldbus" is needed
   // "SETPOINT_APPLICATION_MODE": Operating_Mode: 10x: Jog; 30x: Ref.; 40x: Pos.; 700: Brake test 
   //     => Manual "MOVIKIT® Positioning, Velocity"
   // "TARGET_POSITION":	Target Position in user unit (DINT)
   // 
   // Outputs of the FC:
   // 
   // If the data transmission/PROFINET is disrupted, all outputs will be deleted..
   // => "COMMUNICATION_OK = false (self-confirming)
   // "READY" = true: Ready for operation.
   // "STO_INACTIVE" = true: STO inactive.
   // "OUTPUT_STAGE_ENABLED" = true: Output stage enabled.
   // "BRAKE_RELEASED" = true: Brake released.
   // "MOTOR_TURNING" = true: Motor running
   // "ACTIVE_DRIVE_REFERENCED" = true: Active drive referenced
   // "NEW_RELATIVE_POSITION_APPLIED" = true: New relative position applied
   // "IN_POSITION_SIGNAL_ACTIVE" = true: "In position" signal active
   // "FAULT" = true: Fault.
   // "WARNING" = true: Warning 
   // "DRIVE_TRAIN_2_ACTIVE" = true: Drive train 2 active.
   // "SETPOINT-ACTUAL_COMPARISON"
   // "SW_LIMIT_SWITCHES_INACTIVE" = true: Software limit switches inactive
   //  "STANDBY_MODE_INACTIVE" = true: Stand-by Mode is active.
   // "HEARTBEAT_OUT" : This signal is copied internally from "HEARTBEAT_IN"
   // "ACTUAL_SPEED": in user unit (INT) 
   // "STATUS_MAIN_FAULT_SUB_FAULT:" (WORD)
   //    No fault: Display of current FCB; fault/warning:  High-Byte Fault; Low-Byte SubFault
   // "ACTUAL_TORQUE":in user unit (INT)
   // "DIGITAL_INPUTS" : The digital inputs are read out
   // "ACTUAL_APPLICATION_MODE":	Actual Operating_Mode: 10x: Jog; 30x: Ref.; 40x: Pos.; 700: Brake test 
   //     => Manual "MOVIKIT® Positioning, Velocity"
   // "ACTUAL_POSITION":	 Actual Position in user unit (DINT)
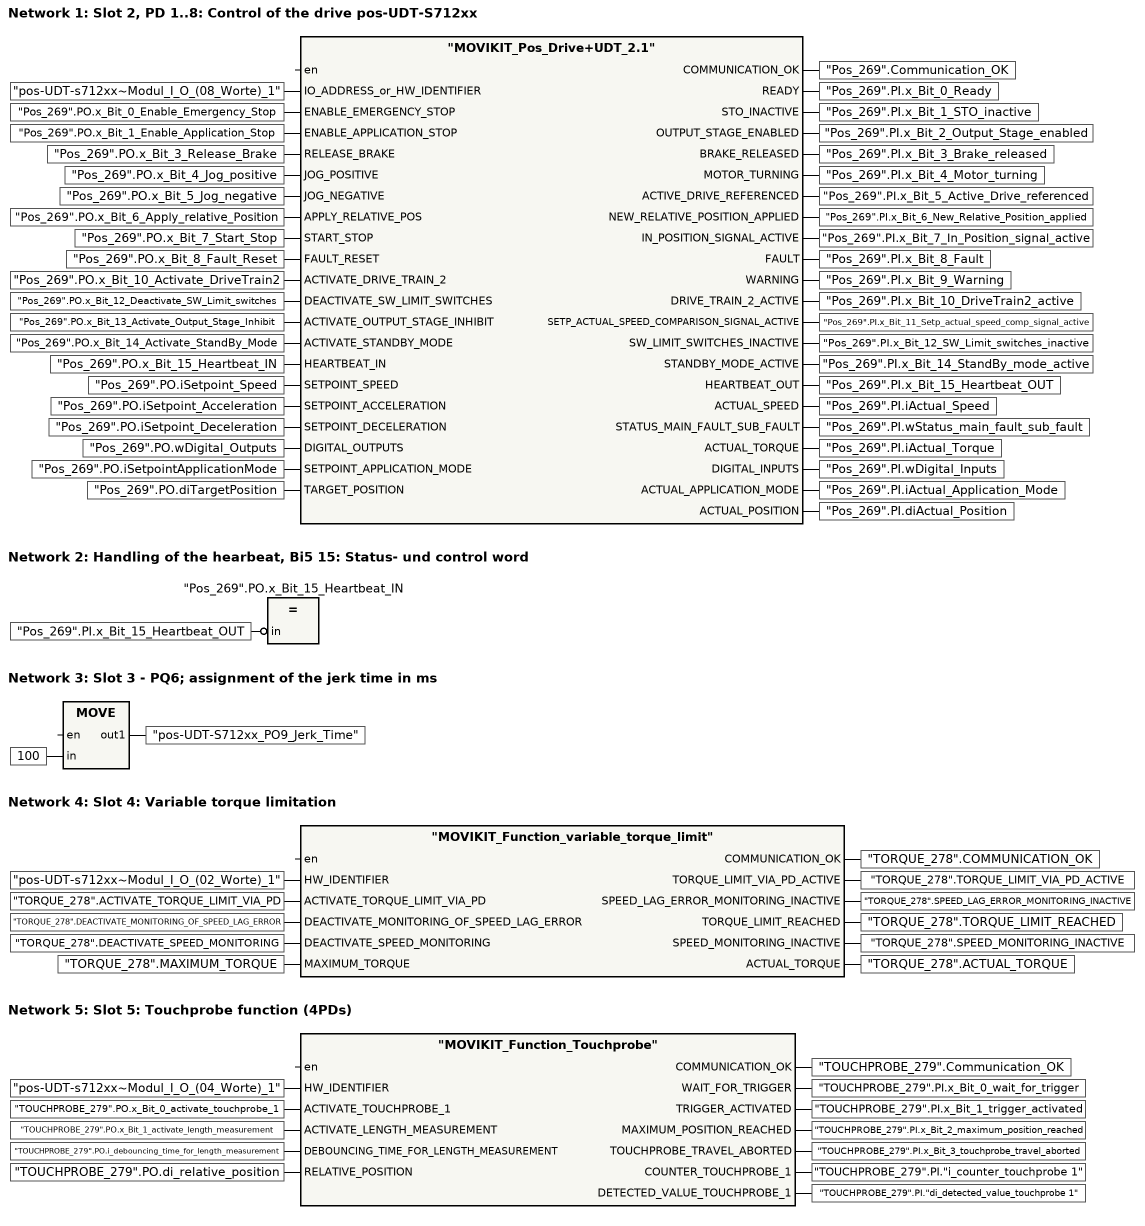
   "MOVIKIT_Pos_Drive+UDT_2.1"(IO_ADDRESS_or_HW_IDENTIFIER := "pos-UDT-s712xx~Modul_I_O_(08_Worte)_1",
                           ENABLE_EMERGENCY_STOP := "Pos_269".PO.x_Bit_0_Enable_Emergency_Stop,
                           ENABLE_APPLICATION_STOP := "Pos_269".PO.x_Bit_1_Enable_Application_Stop,
                           RELEASE_BRAKE := "Pos_269".PO.x_Bit_3_Release_Brake,
                           JOG_POSITIVE := "Pos_269".PO.x_Bit_4_Jog_positive,
                           JOG_NEGATIVE := "Pos_269".PO.x_Bit_5_Jog_negative,
                           APPLY_RELATIVE_POS := "Pos_269".PO.x_Bit_6_Apply_relative_Position,
                           START_STOP := "Pos_269".PO.x_Bit_7_Start_Stop,
                           FAULT_RESET := "Pos_269".PO.x_Bit_8_Fault_Reset,
                           ACTIVATE_DRIVE_TRAIN_2 := "Pos_269".PO.x_Bit_10_Activate_DriveTrain2,
                           DEACTIVATE_SW_LIMIT_SWITCHES := "Pos_269".PO.x_Bit_12_Deactivate_SW_Limit_switches,
                           ACTIVATE_OUTPUT_STAGE_INHIBIT := "Pos_269".PO.x_Bit_13_Activate_Output_Stage_Inhibit,
                           ACTIVATE_STANDBY_MODE := "Pos_269".PO.x_Bit_14_Activate_StandBy_Mode,
                           HEARTBEAT_IN := "Pos_269".PO.x_Bit_15_Heartbeat_IN,
                           SETPOINT_SPEED := "Pos_269".PO.iSetpoint_Speed,
                           SETPOINT_ACCELERATION := "Pos_269".PO.iSetpoint_Acceleration,
                           SETPOINT_DECELERATION := "Pos_269".PO.iSetpoint_Deceleration,
                           DIGITAL_OUTPUTS := "Pos_269".PO.wDigital_Outputs,
                           SETPOINT_APPLICATION_MODE := "Pos_269".PO.iSetpointApplicationMode,
                           TARGET_POSITION := "Pos_269".PO.diTargetPosition,
                           COMMUNICATION_OK => "Pos_269".Communication_OK,
                           READY => "Pos_269".PI.x_Bit_0_Ready,
                           STO_INACTIVE => "Pos_269".PI.x_Bit_1_STO_inactive,
                           OUTPUT_STAGE_ENABLED => "Pos_269".PI.x_Bit_2_Output_Stage_enabled,
                           BRAKE_RELEASED => "Pos_269".PI.x_Bit_3_Brake_released,
                           MOTOR_TURNING => "Pos_269".PI.x_Bit_4_Motor_turning,
                           ACTIVE_DRIVE_REFERENCED => "Pos_269".PI.x_Bit_5_Active_Drive_referenced,
                           NEW_RELATIVE_POSITION_APPLIED => "Pos_269".PI.x_Bit_6_New_Relative_Position_applied,
                           IN_POSITION_SIGNAL_ACTIVE => "Pos_269".PI.x_Bit_7_In_Position_signal_active,
                           FAULT => "Pos_269".PI.x_Bit_8_Fault,
                           WARNING => "Pos_269".PI.x_Bit_9_Warning,
                           DRIVE_TRAIN_2_ACTIVE => "Pos_269".PI.x_Bit_10_DriveTrain2_active,
                           SETP_ACTUAL_SPEED_COMPARISON_SIGNAL_ACTIVE => "Pos_269".PI.x_Bit_11_Setp_actual_speed_comp_signal_active,
                           SW_LIMIT_SWITCHES_INACTIVE => "Pos_269".PI.x_Bit_12_SW_Limit_switches_inactive,
                           STANDBY_MODE_ACTIVE => "Pos_269".PI.x_Bit_14_StandBy_mode_active,
                           HEARTBEAT_OUT => "Pos_269".PI.x_Bit_15_Heartbeat_OUT,
                           ACTUAL_SPEED => "Pos_269".PI.iActual_Speed,
                           STATUS_MAIN_FAULT_SUB_FAULT => "Pos_269".PI.wStatus_main_fault_sub_fault,
                           ACTUAL_TORQUE => "Pos_269".PI.iActual_Torque,
                           DIGITAL_INPUTS => "Pos_269".PI.wDigital_Inputs,
                           ACTUAL_APPLICATION_MODE => "Pos_269".PI.iActual_Application_Mode,
                           ACTUAL_POSITION => "Pos_269".PI.diActual_Position);
END_REGION

REGION Network 2: Handling of the hearbeat, Bi5 15: Status- und control word
   "Pos_269".PO.x_Bit_15_Heartbeat_IN := NOT "Pos_269".PI.x_Bit_15_Heartbeat_OUT;
END_REGION

REGION Network 3: Slot 3 - PQ6; assignment of the jerk time in ms
   // This additional function extends the range of functions
   // by providing the ability to specify the jerk time.
   // The additional function extends the process data
   // length by one process data word.
   // 
   // The jerk is written directly on the output word:
   "pos-UDT-S712xx_PO9_Jerk_Time" := 100;
END_REGION

REGION Network 4: Slot 4: Variable torque limitation
   // The additional function "Variable torque limiting Q1" lets you specify the torque via the
   // application in 0.1% × nominal motor torque. For fieldbus
   // operation, the process data length is extended by 2 process data words.
   // 
   // Inputs of the FC:
   // 
   // Attention! 
   // S71xxx: "HW_Identifier". Assign the HW-Identifier of the 2 PD slot. 
   // S73xx/4xx:"HW_Identifier"Change the data type from "HW_IO" to "WORD" Assign the peripheral address of the 2 PD slot;
   // 
   // "ACTIVATE_TORQUE_LIMIT_VIA_PD": Activation of torque limiting
   // "DEACTIVATE_MONITORING_OF_SPEED_LAG_ERROR": Deactivation of monitoring for speed and lag error
   // "DEACTIVATE_SPEED_MONITORING": Deactivation of speed monitoring
   // "MAXIMUM_TORQUE": Torque related to the nominal motor torque (unit: 0.1%)
   // 
   // Outputs of the FC:
   // 
   // If the data transmission/PROFINET is disrupted, all outputs will be deleted..
   // => "COMMUNICATION_OK = false (self-confirming)
   // "TORQUE_LIMIT_VIA_PD_ACTIVE": Torque limit via PD active
   // "SPEED_LAG_ERROR_MONITORING_INACTIVE": Speed and lag error inactive
   // "TORQUE_LIMIT_REACHED": Torque limit reached
   // "SPEED_MONITORING_INACTIVE": Speed monitoring inactive
   // "ACTUAL_TORQUE": Current torque in relation to the nominal motor torque (unit: 0.1%)
   "MOVIKIT_Function_variable_torque_limit"(HW_IDENTIFIER := "pos-UDT-s712xx~Modul_I_O_(02_Worte)_1",
                           ACTIVATE_TORQUE_LIMIT_VIA_PD := "TORQUE_278".ACTIVATE_TORQUE_LIMIT_VIA_PD,
                           DEACTIVATE_MONITORING_OF_SPEED_LAG_ERROR := "TORQUE_278".DEACTIVATE_MONITORING_OF_SPEED_LAG_ERROR,
                           DEACTIVATE_SPEED_MONITORING := "TORQUE_278".DEACTIVATE_SPEED_MONITORING,
                           MAXIMUM_TORQUE := "TORQUE_278".MAXIMUM_TORQUE,
                           COMMUNICATION_OK => "TORQUE_278".COMMUNICATION_OK,
                           TORQUE_LIMIT_VIA_PD_ACTIVE => "TORQUE_278".TORQUE_LIMIT_VIA_PD_ACTIVE,
                           SPEED_LAG_ERROR_MONITORING_INACTIVE => "TORQUE_278".SPEED_LAG_ERROR_MONITORING_INACTIVE,
                           TORQUE_LIMIT_REACHED => "TORQUE_278".TORQUE_LIMIT_REACHED,
                           SPEED_MONITORING_INACTIVE => "TORQUE_278".SPEED_MONITORING_INACTIVE,
                           ACTUAL_TORQUE => "TORQUE_278".ACTUAL_TORQUE);
END_REGION

REGION Network 5: Slot 5: Touchprobe function (4PDs)
   // => The process data length is extended by 2 process data words.
   "MOVIKIT_Function_Touchprobe"(HW_IDENTIFIER := "pos-UDT-s712xx~Modul_I_O_(04_Worte)_1",
                           ACTIVATE_TOUCHPROBE_1 := "TOUCHPROBE_279".PO.x_Bit_0_activate_touchprobe_1,
                           ACTIVATE_LENGTH_MEASUREMENT := "TOUCHPROBE_279".PO.x_Bit_1_activate_length_measurement,
                           DEBOUNCING_TIME_FOR_LENGTH_MEASUREMENT := "TOUCHPROBE_279".PO.i_debouncing_time_for_length_measurement,
                           RELATIVE_POSITION := "TOUCHPROBE_279".PO.di_relative_position,
                           COMMUNICATION_OK => "TOUCHPROBE_279".Communication_OK,
                           WAIT_FOR_TRIGGER => "TOUCHPROBE_279".PI.x_Bit_0_wait_for_trigger,
                           TRIGGER_ACTIVATED => "TOUCHPROBE_279".PI.x_Bit_1_trigger_activated,
                           MAXIMUM_POSITION_REACHED => "TOUCHPROBE_279".PI.x_Bit_2_maximum_position_reached,
                           TOUCHPROBE_TRAVEL_ABORTED => "TOUCHPROBE_279".PI.x_Bit_3_touchprobe_travel_aborted,
                           COUNTER_TOUCHPROBE_1 => "TOUCHPROBE_279".PI."i_counter_touchprobe 1",
                           DETECTED_VALUE_TOUCHPROBE_1 => "TOUCHPROBE_279".PI."di_detected_value_touchprobe 1");
END_REGION
END_FUNCTION

FUNCTION "MOVIKIT _Positioning_ Drive_2.1" : Void   // FC140, SCL
TITLE = MOVIKIT _Positioning_ Drive
{ S7_Optimized_Access := 'TRUE' }
AUTHOR : CSCEASDI
FAMILY : MOVIKIT
VERSION : 2.1
// This sample program only demonstrates the basic approach. We do not accept any legal or other liability for incorrect program functions and their consequences!
// 
// The FC140 serves as a program module for controlling the MOVIKIT module "Positioning Drive" for the Generation C device series. With the help of the FC140,
// the converters can be controlled via PROFINET IO/PROFIBUS DP.
// 
// Device & networks: To use this FC, a 8 PD slot must be configured.
// 
// Attention Input "HW_Identifier":
// Assign the HW-Identifier of the 8 PD slot.
   VAR_INPUT
      HW_IDENTIFIER : Hw_Io;   // S71xxx: Assign the HW-Identifier of the 8 PD slot.
      ENABLE_EMERGENCY_STOP : Bool;   // true: Enable; false: emergency stop
      ENABLE_APPLIKATION_STOP : Bool;   // true: Enable; false: Application stop
      RELEASE_BRAKE : Bool;   // true: release brake (without enable)
      JOG_POSITIVE : Bool;   // true: Jog positive
      JOG_NEGATIVE : Bool;   // true: Jog negative
      APPLY_RELATIVE_POSITION : Bool;   // true: Apply relative position
      START_STOP : Bool;   // Start/stop with fieldbus ramp
      FAULT_RESET : Bool;   // true: Fault reset
      ACTIVATE_DRIVE_TRAIN_2 : Bool;   // true: Activate drive train 2
      DEACTIVATE_SW_LIMIT_SWITCHES : Bool;   // true: Deactivate software limit switches
      ACTIVATE_OUTPUT_STAGE_INHIBIT : Bool;   // true: Activate output stage inhibit
      ACTIVATE_STANDBY_MODE : Bool;   // true: Activate standby mode
      HEARBEAT_IN : Bool;   // Copied to HEARTBEAT_OUT
      SETPOINT_SPEED : Int;   // in user unit (INT)
      SETPOINT_ACCELERATION : Int;   // in user unit (INT)
      SETPOINT_DECELERATION : Int;   // in user unit (INT)
      DIGITAL_OUTPUTS : Word;   // MoviSuite/Movikit../Inputs/Outputs: dig Outputs: the setting "control via fieldbus" is needed
      SETPOINT_APPLICATION_MODE : Int;   // Operating_Mode: 10x: Jog; 30x: Ref.; 40x: Pos.; 700: Brake test => Manual "MOVIKIT® Positioning, Velocity"
      TARGET_POSITION : DInt;   // Target Position in user unit
   END_VAR
   VAR_OUTPUT
      COMMUNICATION_OK : Bool;   // true: DPRD_DAT and DPWR_DAT are working correctly. false: 5 PD slot required; Check input "HW_Identifier
      READY : Bool;   // true: Ready for operation.
      STO_INACTIVE : Bool;   // true: STO inactive.
      OUTPUT_STAGE_ENABLED : Bool;   // true: Output stage enabled.
      BRAKE_RELEASED : Bool;   // true: Brake released.
      MOTOR_TURNING : Bool;   // true: Motor turning.
      ACTIVE_DRIVE_REFERENCED : Bool;   // true: Active drive referenced
      NEW_RELATIVE_POSITION_APPLIED : Bool;   // true: New relative position applied
      IN_POSITION_SIGNAL_ACTIVE : Bool;   // true: "In position" signal active
      FAULT : Bool;   // true: Fault.
      WARNING : Bool;   // true: Warning
      DRIVE_TRAIN_2_ACTIVE : Bool;   // true: Drive train 2 active.
      SETP_ACTUAL_SPEED_COMPARISON_SIGNAL_ACTIVE : Bool;
      SW_LIMIT_SWITCHES_INACTIVE : Bool;   // true: Software limit switches inactive
      STANDBY_MODE_ACTIVE : Bool;   // true: Stand-by Mode is active.
      HEARTBEAT_OUT : Bool;   // This signal is copied internally from "HEARTBEAT_IN"
      ACTUAL_SPEED : Int;   // in user unit (INT)
      STATUS_MAIN_FAULT_SUB_FAULT : Word;   // No fault: Display of current FCB; fault/warning: High-Byte Fault; Low-Byte SubFault
      ACTUAL_TORQUE : Int;   // in user unit (INT)
      DIGITAL_INPUTS : Word;   // The digital inputs are read out
      ACTUAL_APPLICATION_MODE : Int;   // Actual Operating_Mode: 10x: Jog; 30x: Ref.; 40x: Pos.; 700: Brake test => Manual "MOVIKIT® Positioning, Velocity"
      ACTUAL_POSITION : DInt;   // Actual Position in user unit
   END_VAR
   VAR_TEMP
      PI : Array[1..8] of Word;
      PO : Array[1..8] of Word;
      DPRD_RET_VAL : Int;
      DPWR_RET_VAL : Int;
   END_VAR
BEGIN
   (*This sample program only demonstrates the basic approach. We do not accept any legal or other liability for incorrect program functions and their consequences!

   The FC140 serves as a program module for controlling the MOVIKIT module "Positioning Drive" for the Generation C device series. With the help of the FC140,
   the converters can be controlled via PROFINET IO/PROFIBUS DP.

   Device & networks: To use this FC, a 8 PD slot must be configured.

   Attention Input "HW_Identifier":
   Assign the HW-Identifier of the 8 PD slot. 
   *)

   //DPRD_DAT: Reading Consistent Data of a DP Standard Slave/PROFINET IO device
   #DPRD_RET_VAL:=DPRD_DAT(LADDR:=#HW_IDENTIFIER, RECORD=>#PI);


   IF #DPRD_RET_VAL = 0 THEN //If no error occurs while the instruction is being executed...
       #COMMUNICATION_OK := TRUE;

       //Mapping the signals of the Status word:
       #READY := #PI[1].%X0;
       #STO_INACTIVE := #PI[1].%X1;
       #OUTPUT_STAGE_ENABLED := #PI[1].%X2;
       #BRAKE_RELEASED := #PI[1].%X3;
       #MOTOR_TURNING := #PI[1].%X4;
       #ACTIVE_DRIVE_REFERENCED := #PI[1].%X5;
       #NEW_RELATIVE_POSITION_APPLIED := #PI[1].%X6;
       #IN_POSITION_SIGNAL_ACTIVE := #PI[1].%X7;
       #FAULT := #PI[1].%X8;
       #WARNING := #PI[1].%X9;
       #DRIVE_TRAIN_2_ACTIVE := #PI[1].%X10;
       #SETP_ACTUAL_SPEED_COMPARISON_SIGNAL_ACTIVE := #PI[1].%X11;
       #SW_LIMIT_SWITCHES_INACTIVE:= #PI[1].%X12;
       #STANDBY_MODE_ACTIVE := #PI[1].%X14;
       #HEARTBEAT_OUT := #PI[1].%X15;

       //Assign PI2..8
       #ACTUAL_SPEED := WORD_TO_INT(#PI[2]);
       #STATUS_MAIN_FAULT_SUB_FAULT := #PI[3];
       #ACTUAL_TORQUE := WORD_TO_INT(#PI[4]);
       #DIGITAL_INPUTS := #PI[5];
       #ACTUAL_APPLICATION_MODE := WORD_TO_INT(#PI[6]);
       #ACTUAL_POSITION := SHL(IN := WORD_TO_DINT(#PI[7]), N := 16) + WORD_TO_DINT(#PI[8]);

       //Mapping the signals of the control word:
       #PO[1].%X0 := #ENABLE_EMERGENCY_STOP;
       #PO[1].%X1 := #ENABLE_APPLIKATION_STOP;
       #PO[1].%X3 := #RELEASE_BRAKE;
       #PO[1].%X4 := #JOG_POSITIVE;
       #PO[1].%X5 := #JOG_NEGATIVE;
       #PO[1].%X6 := #APPLY_RELATIVE_POSITION;
       #PO[1].%X7 := #START_STOP;
       #PO[1].%X8 := #FAULT_RESET;
       #PO[1].%X10 := #ACTIVATE_DRIVE_TRAIN_2;
       #PO[1].%X12 := #DEACTIVATE_SW_LIMIT_SWITCHES;
       #PO[1].%X13 := #ACTIVATE_OUTPUT_STAGE_INHIBIT;
       #PO[1].%X14 := #ACTIVATE_STANDBY_MODE;
       #PO[1].%X15 := #HEARBEAT_IN;

       //Set the not used Bits to "false"
       #PO[1].%X2 := FALSE;
       #PO[1].%X9 := FALSE;
       #PO[1].%X11 := FALSE;

       //Assig the POs 2..8
       #PO[2] := INT_TO_WORD(#SETPOINT_SPEED);
       #PO[3] := INT_TO_WORD(#SETPOINT_ACCELERATION);
       #PO[4] := INT_TO_WORD(#SETPOINT_DECELERATION);
       #PO[5] := #DIGITAL_OUTPUTS;
       #PO[6] := INT_TO_WORD(#SETPOINT_APPLICATION_MODE);
       #PO[7] := DINT_TO_WORD(SHR(IN :=#TARGET_POSITION, N := 16));
       #PO[8] := DINT_TO_WORD(#TARGET_POSITION);

   ELSE
       GOTO END;
   END_IF;

   //DPWR_DAT: Write consistent data of a DP standard slave/PROFINET IO device
   #DPWR_RET_VAL := DPWR_DAT(LADDR := #HW_IDENTIFIER, RECORD := #PO);

   END:
   IF #DPRD_RET_VAL <> 0 OR #DPWR_RET_VAL <> 0 THEN
       #COMMUNICATION_OK := FALSE;
       //Erase FC outputs in case of an error
       #READY := FALSE;
       #STO_INACTIVE := FALSE;
       #OUTPUT_STAGE_ENABLED := FALSE;
       #BRAKE_RELEASED := FALSE;
       #MOTOR_TURNING := FALSE;
       #ACTIVE_DRIVE_REFERENCED := FALSE;
       #NEW_RELATIVE_POSITION_APPLIED := FALSE;
       #IN_POSITION_SIGNAL_ACTIVE := FALSE;
       #FAULT := FALSE;
       #WARNING := FALSE;
       #DRIVE_TRAIN_2_ACTIVE := FALSE;
       #SETP_ACTUAL_SPEED_COMPARISON_SIGNAL_ACTIVE := FALSE;
       #SW_LIMIT_SWITCHES_INACTIVE := FALSE;
       #STANDBY_MODE_ACTIVE := FALSE;
       #HEARTBEAT_OUT := FALSE;
       #ACTUAL_SPEED := 0;
       #STATUS_MAIN_FAULT_SUB_FAULT := 0;
       #ACTUAL_TORQUE := 0;
       #DIGITAL_INPUTS := 0;
       #ACTUAL_APPLICATION_MODE := 0;
       #ACTUAL_POSITION := 0;

   END_IF;
END_FUNCTION

FUNCTION "MOVIKIT_Pos_Drive+UDT_2.1" : Void   // FC141, SCL
TITLE = Movikit_Pos_Drive+UDT
{ S7_Optimized_Access := 'FALSE' }
AUTHOR : CSCEASDI
FAMILY : MOVIKIT
VERSION : 2.1
// This sample program only demonstrates the basic approach. We do not accept any legal or other liability for incorrect program functions and their consequences!
// 
// The FC141 serves as a program module for controlling the MOVIKIT module "Positioning Drive+UDT" for the Generation C device series. With the help of the FC141,
// the converters can be controlled via PROFINET IO/PROFIBUS DP.
// 
// Device & networks: To use this FC, a 8 PD slot must be configured.
// 
// This FC uses the UDTs SEW_MOVIKIT_PositioningDrive_SETPOINTS_V2.1 and SEW_MOVIKIT_PositioningDriveDrive_STATUS_V2.1. 
// Please make sure that these PLC data types are available in your TIA project.
// These UDTs can be copied from the original TIA sample project or from the MOVIKIT_Vel_&_Pos_UDTs_V2.1.al14 library.
// 
// Attention Input "HW_Identifier":
// Assign the HW-Identifier of the 8 PD slot. S73xx/4xx:Change Data type from HW_IO to WORD;  Assign the peripheral address of the 8 PD slot
   VAR_INPUT
      IO_ADDRESS_or_HW_IDENTIFIER : Hw_Io;   // S71xxx: Assign the HW-Identifier of the 5 PD slot. S73xx/4xx:Change Data type from HW_IO to WORD; Assign the peripheral address of the 8 PD slot
      ENABLE_EMERGENCY_STOP : Bool;   // true: Enable; false: emergency stop
      ENABLE_APPLICATION_STOP : Bool;   // true: Enable; false: Application stop
      RELEASE_BRAKE : Bool;   // true: release brake (without enable)
      JOG_POSITIVE : Bool;   // true: Jog positive
      JOG_NEGATIVE : Bool;   // true: Jog negative
      APPLY_RELATIVE_POS : Bool;   // true: Apply relative position
      START_STOP : Bool;   // Start/stop with fieldbus ramp
      FAULT_RESET : Bool;   // true: Fault reset
      ACTIVATE_DRIVE_TRAIN_2 : Bool;   // true: Activate drive train 2
      DEACTIVATE_SW_LIMIT_SWITCHES : Bool;   // true: Deactivate software limit switches
      ACTIVATE_OUTPUT_STAGE_INHIBIT : Bool;   // true: Activate output stage inhibit
      ACTIVATE_STANDBY_MODE : Bool;   // true: Activate standby mode
      HEARTBEAT_IN : Bool;   // Copied to HEARTBEAT_OUT
      SETPOINT_SPEED : Int;   // in user unit (INT)
      SETPOINT_ACCELERATION : Int;   // in user unit (INT)
      SETPOINT_DECELERATION : Int;   // in user unit (INT)
      DIGITAL_OUTPUTS : Word;   // MoviSuite/Movikit../Inputs/Outputs: dig Outputs: the setting "control via fieldbus" is needed
      SETPOINT_APPLICATION_MODE : Int;   // Operating_Mode: 10x: Jog; 30x: Ref.; 40x: Pos.; 700: Brake test => Manual "MOVIKIT® Positioning, Velocity"
      TARGET_POSITION : DInt;   // Target Position in user unit
   END_VAR
   VAR_OUTPUT
      COMMUNICATION_OK : Bool;   // true: DPRD_DAT and DPWR_DAT are working correctly. false: 5 PD slot required; Check input "HW_Identifier"
      READY : Bool;   // true: Ready for operation.
      STO_INACTIVE : Bool;   // true: STO inactive.
      OUTPUT_STAGE_ENABLED : Bool;   // true: Output stage enabled.
      BRAKE_RELEASED : Bool;   // true: Brake released.
      MOTOR_TURNING : Bool;   // true: Motor turning.
      ACTIVE_DRIVE_REFERENCED : Bool;   // true: Active drive referenced
      NEW_RELATIVE_POSITION_APPLIED : Bool;   // true: New relative position applied
      IN_POSITION_SIGNAL_ACTIVE : Bool;   // true: "In position" signal active
      FAULT : Bool;   // true: Fault.
      WARNING : Bool;   // true: Warning
      DRIVE_TRAIN_2_ACTIVE : Bool;   // true: Drive train 2 active.
      SETP_ACTUAL_SPEED_COMPARISON_SIGNAL_ACTIVE : Bool;
      SW_LIMIT_SWITCHES_INACTIVE : Bool;   // true: Software limit switches inactive
      STANDBY_MODE_ACTIVE : Bool;   // true: Stand-by Mode is active.
      HEARTBEAT_OUT : Bool;   // This signal is copied internally from "HEARTBEAT_IN"
      ACTUAL_SPEED : Int;   // in user unit (INT)
      STATUS_MAIN_FAULT_SUB_FAULT : Word;   // No fault: Display of current FCB; fault/warning: High-Byte Fault; Low-Byte SubFault
      ACTUAL_TORQUE : Int;   // in user unit (INT)
      DIGITAL_INPUTS : Word;   // The digital inputs are read out
      ACTUAL_APPLICATION_MODE : Int;   // Actual Operating_Mode: 10x: Jog; 30x: Ref.; 40x: Pos.; 700: Brake test => Manual "MOVIKIT® Positioning, Velocity"
      ACTUAL_POSITION : DInt;   // Actual Position in user unit
   END_VAR
   VAR_TEMP
      PI : "SEW_MOVIKIT_PositioningDrive_STATUS_V2.1";
      PO : "SEW_MOVIKIT_PositioningDrive_SETPOINTS_V2.1";
      DPRD_RET_VAL : Int;
      DPWR_RET_VAL : Int;
   END_VAR
BEGIN
   (*This sample program only demonstrates the basic approach. We do not accept any legal or other liability for incorrect program functions and their consequences!

   The FC141 serves as a program module for controlling the MOVIKIT module "Positioning Drive+UDT" for the Generation C device series. With the help of the FC141,
   the converters can be controlled via PROFINET IO/PROFIBUS DP.

   Device & networks: To use this FC, a 8 PD slot must be configured.

   This FC uses the UDTs SEW_MOVIKIT_PositioningDrive_SETPOINTS_V2.1 and SEW_MOVIKIT_PositioningDriveDrive_STATUS_V2.1. 
   Please make sure that these PLC data types are available in your TIA project.
   These UDTs can be copied from the original TIA sample project or from the MOVIKIT_Vel_&_Pos_UDTs_V2.x.al14 library.

   Attention Input "HW_Identifier":
   Assign the HW-Identifier of the 8 PD slot. S73xx/4xx:Change Data type from HW_IO to WORD;  Assign the peripheral address of the 8 PD slot
   *)

   //DPRD_DAT: Reading Consistent Data of a DP Standard Slave/PROFINET IO device
   #DPRD_RET_VAL := DPRD_DAT(LADDR := #IO_ADDRESS_or_HW_IDENTIFIER, RECORD => #PI);


   IF #DPRD_RET_VAL = 0 THEN //If no error occurs while the instruction is being executed...
       #COMMUNICATION_OK := TRUE;

       //Mapping the signals of the Status word:
       #READY := #PI.x_Bit_0_Ready;
       #STO_INACTIVE := #PI.x_Bit_1_STO_inactive;
       #OUTPUT_STAGE_ENABLED := #PI.x_Bit_2_Output_Stage_enabled;
       #BRAKE_RELEASED := #PI.x_Bit_3_Brake_released;
       #MOTOR_TURNING := #PI.x_Bit_4_Motor_turning;
       #ACTIVE_DRIVE_REFERENCED := #PI.x_Bit_5_Active_Drive_referenced;
       #NEW_RELATIVE_POSITION_APPLIED := #PI.x_Bit_6_New_Relative_Position_applied;
       #IN_POSITION_SIGNAL_ACTIVE := #PI.x_Bit_7_In_Position_signal_active;
       #FAULT := #PI.x_Bit_8_Fault;
       #WARNING := #PI.x_Bit_9_Warning;
       #DRIVE_TRAIN_2_ACTIVE := #PI.x_Bit_10_DriveTrain2_active;
       #SETP_ACTUAL_SPEED_COMPARISON_SIGNAL_ACTIVE := #PI.x_Bit_11_Setp_actual_speed_comp_signal_active;
       #SW_LIMIT_SWITCHES_INACTIVE:= #PI.x_Bit_12_SW_Limit_switches_inactive;
       #STANDBY_MODE_ACTIVE := #PI.x_Bit_14_StandBy_mode_active;
       #HEARTBEAT_OUT := #PI.x_Bit_15_Heartbeat_OUT;

       //Assign PI2..8
       #ACTUAL_SPEED := #PI.iActual_Speed;
       #STATUS_MAIN_FAULT_SUB_FAULT := #PI.wStatus_main_fault_sub_fault;
       #ACTUAL_TORQUE := #PI.iActual_Torque;
       #DIGITAL_INPUTS := #PI.wDigital_Inputs;
       #ACTUAL_APPLICATION_MODE := #PI.iActual_Application_Mode;
       #ACTUAL_POSITION := #PI.diActual_Position;

       //Mapping the signals of the control word:
       #PO.x_Bit_0_Enable_Emergency_Stop := #ENABLE_EMERGENCY_STOP;
       #PO.x_Bit_1_Enable_Application_Stop := #ENABLE_APPLICATION_STOP;
       #PO.x_Bit_3_Release_Brake := #RELEASE_BRAKE;
       #PO.x_Bit_4_Jog_positive := #JOG_POSITIVE;
       #PO.x_Bit_5_Jog_negative := #JOG_NEGATIVE;
       #PO.x_Bit_6_Apply_relative_Position := #APPLY_RELATIVE_POS;;
       #PO.x_Bit_7_Start_Stop := #START_STOP;
       #PO.x_Bit_8_Fault_Reset := #FAULT_RESET;
       #PO.x_Bit_10_Activate_DriveTrain2 := #ACTIVATE_DRIVE_TRAIN_2;
       #PO.x_Bit_12_Deactivate_SW_Limit_switches := #DEACTIVATE_SW_LIMIT_SWITCHES;
       #PO.x_Bit_13_Activate_Output_Stage_Inhibit := #ACTIVATE_OUTPUT_STAGE_INHIBIT;
       #PO.x_Bit_14_Activate_StandBy_Mode := #ACTIVATE_STANDBY_MODE;
       #PO.x_Bit_15_Heartbeat_IN := #HEARTBEAT_IN;


       //Set the not used Bits to "false"
       #PO.x_Bit_2_Reserved := FALSE;
       #PO.x_Bit_9_Reserved := FALSE;
       #PO.x_Bit_11_Reserved := FALSE;

       //Assig the POs 2..8
       #PO.iSetpoint_Speed := #SETPOINT_SPEED;
       #PO.iSetpoint_Acceleration := #SETPOINT_ACCELERATION;
       #PO.iSetpoint_Deceleration := #SETPOINT_DECELERATION;
       #PO.wDigital_Outputs := #DIGITAL_OUTPUTS;
       #PO.iSetpointApplicationMode := #SETPOINT_APPLICATION_MODE;
       #PO.diTargetPosition := #TARGET_POSITION;

   ELSE
       GOTO END;
   END_IF;

   //DPWR_DAT: Write consistent data of a DP standard slave/PROFINET IO device
   #DPWR_RET_VAL := DPWR_DAT(LADDR := #IO_ADDRESS_or_HW_IDENTIFIER, RECORD := #PO);

   END:
   IF #DPRD_RET_VAL <> 0 OR #DPWR_RET_VAL <> 0 THEN
       #COMMUNICATION_OK := FALSE;
       //Erase FC outputs in case of an error
       #READY := FALSE;
       #STO_INACTIVE := FALSE;
       #OUTPUT_STAGE_ENABLED := FALSE;
       #BRAKE_RELEASED := FALSE;
       #MOTOR_TURNING := FALSE;
       #ACTIVE_DRIVE_REFERENCED := FALSE;
       #NEW_RELATIVE_POSITION_APPLIED := FALSE;
       #IN_POSITION_SIGNAL_ACTIVE := FALSE;
       #FAULT := FALSE;
       #WARNING := FALSE;
       #DRIVE_TRAIN_2_ACTIVE := FALSE;
       #SETP_ACTUAL_SPEED_COMPARISON_SIGNAL_ACTIVE := FALSE;
       #SW_LIMIT_SWITCHES_INACTIVE := FALSE;
       #STANDBY_MODE_ACTIVE := FALSE;
       #HEARTBEAT_OUT := FALSE;
       #ACTUAL_SPEED := 0;
       #STATUS_MAIN_FAULT_SUB_FAULT := 0;
       #ACTUAL_TORQUE := 0;
       #DIGITAL_INPUTS := 0;
       #ACTUAL_APPLICATION_MODE := 0;
       #ACTUAL_POSITION := 0;
   END_IF;
END_FUNCTION

FUNCTION "MOVIKIT_Function_variable_torque_limit" : Void   // FC191, SCL
TITLE = Movikit_Function_variable_torque_limit
{ S7_Optimized_Access := 'FALSE' }
AUTHOR : SVSPASE
FAMILY : MOVIKIT
VERSION : 2.0
// This sample program only demonstrates the basic approach. We do not accept any legal or other liability for incorrect program functions and their consequences!
// 
// This FC is used to control the MOVIKIT function "variable torque limit Q1 (2PD)"
// 
// Device & networks: To use this FC, a 2 PD slot must be configured.
// 
// This FC uses the UDTs "SEW_Movikit_Function_torque_limit_SETPOINTS_V1.0" and "SEW_MOVIKIT_Function_torque_limit_STATUS_V1.0". 
// Please make sure that these PLC data types are available in your TIA project.
// These UDTs can be copied from the original TIA sample project or from the MOVIKIT_VELOCITY_UDTs_V1.0.al14 library.
// 
// Attention Input "HW_Identifier":
// Assign the HW-Identifier of the 2 PD slot. S73xx/4xx:Change Data type from HW_IO to WORD;  Assign the peripheral address of the 2 PD slot
   VAR_INPUT
      HW_IDENTIFIER : Hw_Io;   // S71xxx: Assign the HW-Identifier of the 2 PD slot. S73xx/4xx:Change Data type from HW_IO to WORD; Assign the peripheral address of the 2 PD slot
      ACTIVATE_TORQUE_LIMIT_VIA_PD : Bool;   // activate torque limit via PD
      DEACTIVATE_MONITORING_OF_SPEED_LAG_ERROR : Bool;   // deactivate monitoring of lag and speed errors
      DEACTIVATE_SPEED_MONITORING : Bool;   // deactivate speed monitoring
      MAXIMUM_TORQUE : Int;   // maximum torque
   END_VAR
   VAR_OUTPUT
      COMMUNICATION_OK : Bool;
      TORQUE_LIMIT_VIA_PD_ACTIVE : Bool;   // Torque limit via PD active
      SPEED_LAG_ERROR_MONITORING_INACTIVE : Bool;   // Speed and lag error inactive
      TORQUE_LIMIT_REACHED : Bool;   // Torque limit reached
      SPEED_MONITORING_INACTIVE : Bool;   // Speed monitoring inactive
      ACTUAL_TORQUE : Int;   // Actual torque
   END_VAR
   VAR_TEMP
      PI : "SEW_MOVIKIT_Function_torque_limit_STATUS_V2.0";
      PO : "SEW_MOVIKIT_Function_torque_limit_SETPOINTS_V2.0";
      DPRD_RET_VAL : Int;
      DPWR_RET_VAL : Int;
   END_VAR
BEGIN
   (*This sample program only demonstrates the basic approach. We do not accept any legal or other liability for incorrect program functions and their consequences!

   This FC is used to control the MOVIKIT function "variable torque limit Q1 (2PD)"

   Device & networks: To use this FC, a 2 PD slot must be configured.

   This FC uses the UDTs "SEW_Movikit_Function_torque_limit_SETPOINTS_V1.0" and "SEW_MOVIKIT_Function_torque_limit_STATUS_V1.0". 
   Please make sure that these PLC data types are available in your TIA project.
   These UDTs can be copied from the original TIA sample project or from the MOVIKIT_VELOCITY_UDTs_V1.0.al14 library.

   Attention Input "HW_Identifier":
   Assign the HW-Identifier of the 2 PD slot. S73xx/4xx:Change Data type from HW_IO to WORD;  Assign the peripheral address of the 2 PD slot*)



   //DPWR_DAT: Write consistent data of a DP standard slave/PROFINET IO device
   #DPRD_RET_VAL := DPRD_DAT(LADDR := #HW_IDENTIFIER, RECORD => #PI);


   IF #DPRD_RET_VAL = 0 THEN
       #COMMUNICATION_OK := TRUE;

       //Assign the bits of the status word:
       #TORQUE_LIMIT_VIA_PD_ACTIVE := #PI.x_Bit_0_torque_limit_via_PD_active;
       #SPEED_LAG_ERROR_MONITORING_INACTIVE := #PI.x_Bit_1_speed_and_lag_error_monitoring_inactive;
       #TORQUE_LIMIT_REACHED := #PI.x_Bit_2_torque_limit_reached;
       #SPEED_MONITORING_INACTIVE := #PI.x_Bit_3_speed_monitoring_inactive;

       #ACTUAL_TORQUE := #PI.i_actual_torque;

       //Mapping of the process output word:
       #PO.x_Bit_0_activate_torque_limit_via_PD := #ACTIVATE_TORQUE_LIMIT_VIA_PD;
       #PO.x_Bit_1_deactivate_monitoring_of_speed_and_lag_error:= #DEACTIVATE_MONITORING_OF_SPEED_LAG_ERROR;
       #PO.x_Bit_3_deactivate_speed_monitoring := #DEACTIVATE_SPEED_MONITORING;

       //Set the not used Bits to "false"
       #PO.x_Bit_2 := FALSE;
       #PO.x_Bit_4:= FALSE;
       #PO.x_Bit_5:= FALSE;
       #PO.x_Bit_6 := FALSE;
       #PO.x_Bit_7 := FALSE;
       #PO.x_Bit_8 := FALSE;
       #PO.x_Bit_9 := FALSE;
       #PO.x_Bit_10:= FALSE;
       #PO.x_Bit_11:= FALSE;
       #PO.x_Bit_12:= FALSE;
       #PO.x_Bit_13:= FALSE;
       #PO.x_Bit_14:= FALSE;
       #PO.x_Bit_15:= FALSE;

       #PO.i_maximum_torque := #MAXIMUM_TORQUE;

   ELSE
       GOTO END;
   END_IF;

   //DPWR_DAT: Write consistent data of a DP standard slave/PROFINET IO device
   #DPWR_RET_VAL := DPWR_DAT(LADDR := #HW_IDENTIFIER, RECORD := #PO);

   END:
   IF #DPRD_RET_VAL <> 0 OR #DPWR_RET_VAL <> 0 THEN
       #COMMUNICATION_OK := FALSE;

       //Erase FC outputs in case of an error
       #TORQUE_LIMIT_VIA_PD_ACTIVE := FALSE;
       #SPEED_LAG_ERROR_MONITORING_INACTIVE := FALSE;
       #TORQUE_LIMIT_REACHED := FALSE;
       #SPEED_MONITORING_INACTIVE := FALSE;

       #ACTUAL_TORQUE := 0;
   END_IF;
END_FUNCTION

FUNCTION "MOVIKIT_Function_Touchprobe" : Void   // FC192, SCL
TITLE = Movikit_Function_Touchprobe
{ S7_Optimized_Access := 'FALSE' }
AUTHOR : SVSPASE
FAMILY : MOVIKIT
VERSION : 2.0
// This sample program only demonstrates the basic approach. We do not accept any legal or other liability for incorrect program functions and their consequences!
// 
// This FC is used to control the MOVIKIT function "touchprobe"
// 
// Device & networks: To use this FC, a 4 PD slot must be configured.
// 
// This FC uses the UDTs "SEW_Movikit_Function_touchprobe_SETPOINTS_V1.0" and "SEW_MOVIKIT_Function_touchprobe_STATUS_V1.0". 
// Please make sure that these PLC data types are available in your TIA project.
// These UDTs can be copied from the original TIA sample project or from the MOVIKIT_VELOCITY_UDTs_V1.0.al14 library.
// 
// Attention Input "HW_Identifier":
// Assign the HW-Identifier of the 4 PD slot. S73xx/4xx:Change Data type from HW_IO to WORD;  Assign the peripheral address of the 4 PD slot
   VAR_INPUT
      HW_IDENTIFIER : Hw_Io;   // S71xxx: Assign the HW-Identifier of the 2 PD slot. S73xx/4xx:Change Data type from HW_IO to WORD; Assign the peripheral address of the 2 PD slot
      ACTIVATE_TOUCHPROBE_1 : Bool;
      ACTIVATE_LENGTH_MEASUREMENT : Bool;
      DEBOUNCING_TIME_FOR_LENGTH_MEASUREMENT : Int;
      RELATIVE_POSITION : DInt;
   END_VAR
   VAR_OUTPUT
      COMMUNICATION_OK : Bool;
      WAIT_FOR_TRIGGER : Bool;
      TRIGGER_ACTIVATED : Bool;
      MAXIMUM_POSITION_REACHED : Bool;
      TOUCHPROBE_TRAVEL_ABORTED : Bool;
      COUNTER_TOUCHPROBE_1 : Int;
      DETECTED_VALUE_TOUCHPROBE_1 : DInt;
   END_VAR
   VAR_TEMP
      PI : "SEW_MOVIKIT_Function_touchprobe_STATUS_V2.0";
      PO : "SEW_MOVIKIT_Function_touchprobe_SETPOINTS_V2.0";
      DPRD_RET_VAL : Int;
      DPWR_RET_VAL : Int;
   END_VAR
BEGIN
   (*This sample program only demonstrates the basic approach. We do not accept any legal or other liability for incorrect program functions and their consequences!

   This FC is used to control the MOVIKIT function "touchprobe"

   Device & networks: To use this FC, a 4 PD slot must be configured.

   This FC uses the UDTs "SEW_Movikit_Function_touchprobe_SETPOINTS_V1.0" and "SEW_MOVIKIT_Function_touchprobe_STATUS_V1.0". 
   Please make sure that these PLC data types are available in your TIA project.
   These UDTs can be copied from the original TIA sample project or from the MOVIKIT_VELOCITY_UDTs_V1.0.al14 library.

   Attention Input "HW_Identifier":
   Assign the HW-Identifier of the 4 PD slot. S73xx/4xx:Change Data type from HW_IO to WORD;  Assign the peripheral address of the 4 PD slot*)

   //DPWR_DAT: Write consistent data of a DP standard slave/PROFINET IO device
   #DPRD_RET_VAL := DPRD_DAT(LADDR := #HW_IDENTIFIER, RECORD => #PI);

   IF #DPRD_RET_VAL = 0 THEN
       #COMMUNICATION_OK := TRUE;

       //Assign the Bits of the status word
       #WAIT_FOR_TRIGGER:=#PI.x_Bit_0_wait_for_trigger;
       #TRIGGER_ACTIVATED := #PI.x_Bit_1_trigger_activated;
       #MAXIMUM_POSITION_REACHED:= #PI.x_Bit_2_maximum_position_reached;
       #TOUCHPROBE_TRAVEL_ABORTED := #PI.x_Bit_3_touchprobe_travel_aborted;

       //Assign the input words..
       #COUNTER_TOUCHPROBE_1 := #PI."i_counter_touchprobe 1";
       #DETECTED_VALUE_TOUCHPROBE_1 := #PI."di_detected_value_touchprobe 1";

       //Mapping of the status word bits.. 
       #PO.x_Bit_0_activate_touchprobe_1:= #ACTIVATE_TOUCHPROBE_1;
       #PO.x_Bit_1_activate_length_measurement := #ACTIVATE_LENGTH_MEASUREMENT;


       //Set the not used Bits to "false"
       #PO.x_Bit_2 := FALSE;
       #PO.x_Bit_3 := FALSE;
       #PO.x_Bit_4 := FALSE;
       #PO.x_Bit_5 := FALSE;
       #PO.x_Bit_6 := FALSE;
       #PO.x_Bit_7 := FALSE;
       #PO.x_Bit_8 := FALSE;
       #PO.x_Bit_9 := FALSE;
       #PO.x_Bit_10 := FALSE;
       #PO.x_Bit_11 := FALSE;
       #PO.x_Bit_12 := FALSE;
       #PO.x_Bit_13 := FALSE;
       #PO.x_Bit_14 := FALSE;
       #PO.x_Bit_15 := FALSE;

       #PO.i_debouncing_time_for_length_measurement := #DEBOUNCING_TIME_FOR_LENGTH_MEASUREMENT;
       #PO.di_relative_position:=#RELATIVE_POSITION;

   ELSE
       GOTO END;
   END_IF;

   //DPWR_DAT: Write consistent data of a DP standard slave/PROFINET IO device
   #DPWR_RET_VAL := DPWR_DAT(LADDR := #HW_IDENTIFIER, RECORD := #PO);

   END:
   IF #DPRD_RET_VAL <> 0 OR #DPWR_RET_VAL <> 0 THEN
       #COMMUNICATION_OK := FALSE;
       //Erase FC outputs in case of an error
       #COMMUNICATION_OK := false;
       #WAIT_FOR_TRIGGER := false;
       #TRIGGER_ACTIVATED := false;
       #MAXIMUM_POSITION_REACHED := false;
       #TOUCHPROBE_TRAVEL_ABORTED := false;
       #COUNTER_TOUCHPROBE_1 := 0;
       #DETECTED_VALUE_TOUCHPROBE_1:= 0;
   END_IF;
END_FUNCTION

ORGANIZATION_BLOCK "Main"   // OB1, FBD, ProgramCycle
TITLE = "Main Program Sweep (Cycle)"
{ S7_Optimized_Access := 'TRUE' }
VERSION : 0.1
// This sample program only demonstrates the basic approach. We do not accept any legal or other liability for incorrect program functions and their consequences!
// 
// Please take note of the manual "MOVIKIT® Positioning, Velocity"
BEGIN

REGION Network 1: Control of the drive pos-UDT-S712xx with the functions "Variable jerk time, Variable torque limitation, parameter channel via process data (5PD).
   // Control of the drive velocity-UDT-S712xx with the functions "Variable jerk time, Variable torque limitation, parameter channel via process data (5PD).
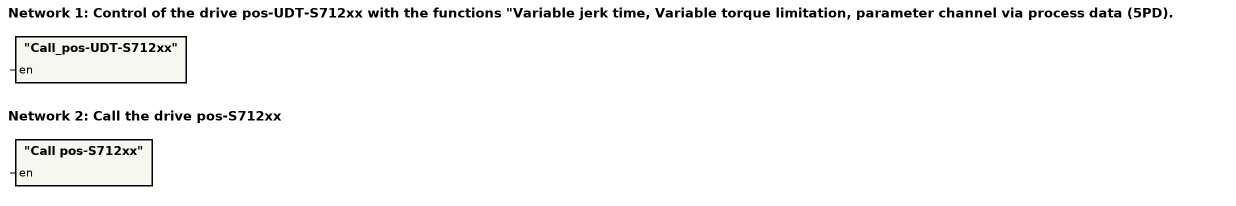
   "Call_pos-UDT-S712xx"();
END_REGION

REGION Network 2: Call the drive pos-S712xx
   // without the use of UDTs, without the functions "Variable jerk time, Variable torque limitation, parameter channel via process data (5PD)
   "Call pos-S712xx"();
END_REGION
END_ORGANIZATION_BLOCK

// ===== PLC "CPU 315F-2 PN/DP"  CPU 315F-2 PN/DP =====

VAR_GLOBAL   // PLC tag table "Standard-Variablentabelle"
   "Clock_0.5Hz" AT %M0.7 : Bool;
   "Clock_Byte" AT %MB0 : Byte;
   "Clock_10Hz" AT %M0.0 : Bool;
   "Clock_5Hz" AT %M0.1 : Bool;
   "Clock_2.5Hz" AT %M0.2 : Bool;
   "Clock_2Hz" AT %M0.3 : Bool;
   "Clock_1.25Hz" AT %M0.4 : Bool;
   "Clock_1Hz" AT %M0.5 : Bool;
   "Clock_0.625Hz" AT %M0.6 : Bool;
   "pos-UDT-S73xx_PO1" AT %AW300 : Word;   // control word
   "pos-UDT-S73xx_PO2" AT %QW302 : Int;   // setpoint speed
   "pos-UDT-S73xx_PO3" AT %QW304 : Int;   // acceleration
   "pos-UDT-S73xx_PO4" AT %QW306 : Int;   // deceleration
   "pos-UDT-S73xx_PO5" AT %QW308 : Word;   // dig. Outputs
   "pos-UDT-S73xx_PI1" AT %IW300 : Word;   // status word
   "pos-UDT-S73xx_PI2" AT %IW302 : Int;   // actual speed
   "pos-UDT-S73xx_PI3" AT %IW304 : Word;   // Status/Main/Subfault
   "pos-UDT-S73xx_PI4" AT %IW306 : Int;   // actual torque
   "pos-UDT-S73xx_PI5" AT %IW308 : Word;   // dig. Inputs
   "pos-UDT-S73xx_PO6" AT %QW310 : Int;   // target application mode
   "pos-UDT-S73xx_PO8" AT %QD312 : DInt;   // target position
   "pos-UDT-S73xx_PI6" AT %IW310 : Int;   // actual application mode
   "pos-UDT-S73xx_PI7-8" AT %ID312 : DInt;   // actual position
END_VAR

TYPE "SEW_MOVIKIT_PositioningDrive_SETPOINTS_V2.1"
TITLE = SEW_MOVIKIT_PositioningDrive_SETPOINTS
// Dieses UDT bildet die 8 Prozeßeingangsdaten des MOVIKIT PositioningDrives ab. This UDT maps the 8 process input data of the MOVIKIT PositioningDrive.
   STRUCT
      x_Bit_8_Fault_Reset : Bool;
      x_Bit_9_Reserved : Bool;
      x_Bit_10_Activate_DriveTrain2 : Bool;
      x_Bit_11_Reserved : Bool;
      x_Bit_12_Deactivate_SW_Limit_switches : Bool;
      x_Bit_13_Activate_Output_Stage_Inhibit : Bool;
      x_Bit_14_Activate_StandBy_Mode : Bool;
      x_Bit_15_Heartbeat_IN : Bool;
      x_Bit_0_Enable_Emergency_Stop : Bool;
      x_Bit_1_Enable_Application_Stop : Bool;
      x_Bit_2_Reserved : Bool;
      x_Bit_3_Release_Brake : Bool;
      x_Bit_4_Jog_positive : Bool;
      x_Bit_5_Jog_negative : Bool;
      x_Bit_6_Apply_relative_Position : Bool;
      x_Bit_7_Start_Stop : Bool;
      iSetpoint_Speed : Int;
      iSetpoint_Acceleration : Int;
      iSetpoint_Deceleration : Int;
      wDigital_Outputs : Word;
      iSetpointApplicationMode : Int;
      diTargetPosition : DInt;
   END_STRUCT;
END_TYPE

TYPE "SEW_MOVIKIT_PositioningDrive_STATUS_V2.1"
TITLE = SEW_MOVIKIT_PositioningDrive_STATUS
// Dieses UDT bildet die 8 Prozeßausgangsdaten des MOVIKIT PositioningDrives ab. This UDT maps the 8 process output data of the MOVIKIT PositioningDrive.
   STRUCT
      x_Bit_8_Fault : Bool;
      x_Bit_9_Warning : Bool;
      x_Bit_10_DriveTrain2_active : Bool;
      x_Bit_11_Setp_actual_speed_comp_signal_active : Bool;
      x_Bit_12_SW_Limit_switches_inactive : Bool;
      x_Bit_13_Reserved : Bool;
      x_Bit_14_StandBy_mode_active : Bool;
      x_Bit_15_Heartbeat_OUT : Bool;
      x_Bit_0_Ready : Bool;
      x_Bit_1_STO_inactive : Bool;
      x_Bit_2_Output_Stage_enabled : Bool;
      x_Bit_3_Brake_released : Bool;
      x_Bit_4_Motor_turning : Bool;
      x_Bit_5_Active_Drive_referenced : Bool;
      x_Bit_6_New_Relative_Position_applied : Bool;
      x_Bit_7_In_Position_signal_active : Bool;
      iActual_Speed : Int;
      wStatus_main_fault_sub_fault : Word;
      iActual_Torque : Int;
      wDigital_Inputs : Word;
      iActual_Application_Mode : Int;
      diActual_Position : DInt;
   END_STRUCT;
END_TYPE

DATA_BLOCK "MOVIKIT_Positioning_256"   // DB256
{ S7_Optimized_Access := 'FALSE' }
VERSION : 0.1
   VAR
      PO : "SEW_MOVIKIT_PositioningDrive_SETPOINTS_V2.1";
      PI : "SEW_MOVIKIT_PositioningDrive_STATUS_V2.1";
      Communication_OK : Bool;   // true: DPRD_DAT and DPWR_DAT are working correctly. false: 5 PD slot required; Check address at Input "IO_ADDRESS"
   END_VAR
BEGIN
END_DATA_BLOCK

DATA_BLOCK "Pos_291"   // DB291
{ S7_Optimized_Access := 'FALSE' }
VERSION : 0.1
   VAR
      ENABLE_EMERGENCY_STOP : Bool;
      ENABLE_APPLICATION_STOP : Bool;
      RELEASE_BRAKE : Bool;
      JOG_POSITIVE : Bool;   // true: Jog positive
      JOG_NEGATIVE : Bool;   // true: Jog negative
      APPLY_RELATIVE_POSITION : Bool;   // true: Apply relative position
      START_STOP : Bool;
      FAULT_RESET : Bool;
      ACTIVATE_DRIVE_TRAIN_2 : Bool;
      DEACTIVATE_SW_LIMIT_SWITCH : Bool;
      ACTIVATE_OUTPUT_STAGE_INHIBIT : Bool;
      ACTIVATE_STANDBY_MODE : Bool;
      HEARTBEAT_IN : Bool;
      SETPOINT_SPEED : Int;
      SETPOINT_ACCELERATION : Int;
      SETPOINT_DECELERATION : Int;
      DIGITAL_OUTPUTS : Word;
      SETPOINT__APPLICATION_MODE : Int;   // Operating_Mode: 10x: Jog; 30x: Ref.; 40x: Pos.; 700: Brake test => Manual "MOVIKIT® Positioning, Velocity"
      TARGET_POSITION : DInt;   // Target Position in user unit
      COMMUNICATION_OK : Bool;
      READY : Bool;
      STO_INACTIVE : Bool;
      OUTPUT_STAGE_ENABLED : Bool;
      BRAKE_RELEASED : Bool;
      MOTOR_TURNING : Bool;
      ACTIVE_DRIVE_REFERENCED : Bool;   // true: Active drive referenced
      NEW_RELATIVE_POSITION_APPLIED : Bool;   // true: New relative position applied
      IN_POSITION_SIGNAL_ACTIVE : Bool;
      FAULT : Bool;
      WARNING : Bool;
      DRIVE_TRAIN_2_ACTIVE : Bool;
      SETP_ACTUAL_SPEED_COMPARISON_SIGNAL_ACTIVE : Bool;
      SW_LIMIT_SWITCH_INACTIVE : Bool;
      STANDBY_MODE_ACTIVE : Bool;
      HEARTBEAT_OUT : Bool;
      ACTUAL_SPEED : Int;
      STATUS_MAIN_FAULT_SUB_FAULT : Int;
      ACTUAL_TORQUE : Int;
      DIGITAL_INPUTS : Word;
      ACTUAL_APPLICATION_MODE : Int;   // Actual Operating_Mode: 10x: Jog; 30x: Ref.; 40x: Pos.; 700: Brake test => Manual "MOVIKIT® Positioning, Velocity"
      ACTUAL_POSITION : DInt;   // Actual Position in user unit
   END_VAR
BEGIN
END_DATA_BLOCK

FUNCTION "Call_pos_UDT_S73xx" : Void   // FC100, FBD
TITLE = Call_pos_UDT_S73xx
{ S7_Optimized_Access := 'FALSE' }
VERSION : 0.1
// This sample program only demonstrates the basic approach. We do not accept any legal or other liability for incorrect program functions and their consequences!
// 
// Please take note of the manual "MOVIKIT® Positioning, Velocity"
BEGIN

REGION Network 1: Control of the drive pos-UDT-S73xx
   // The FC142 serves as a program module for controlling the MOVIKIT module "Positioning Drive" for the Generation C device series. With the help of the FC142, the converters can be controlled via PROFINET IO/PROFIBUS DP. 
   // 
   // Device & networks: To use this FC, a 8 PD slot must be configured.
   // 
   // This FC uses the UDTs "SEW_MOVIKIT_PositioningDrive_SETPOINTS_V2.1" and "SEW_MOVIKIT_PositioningDrive_STATUS_V2.1". Please make sure that these PLC data types are available in your TIA project. These UDTs can be copied from the original TIA sample project or from the MOVIKIT_Positioning_UDTs_V2.x.al14 library.
   // 
   // Inputs of the FC:
   // 
   // Attention! 
   // S73xx/4xx:"IO_ADDRESS"/Data Type Word:  Assign the peripheral address of the 8 PD slot;
   // S71xxx: "IO_ADDRESS" change the data type from Word to "HW_IO". Assign the HW-Identifier of the 8 PD slot. 
   // 
   // "ENABLE_EMERGENCY_STOP" = true: Enable; false: emergency stop
   // "ENABLE_APPLICATION_STOP" = true: Enable; false: Application stop
   // "RELEASE_BRAKE" = true: release brake (without enable)
   // "JOG_POSITIVE": Signal for moving the drive in positive direction in jog mode.
   // "JOG_NEGATIVE": Signal for moving the drive in negative direction in jog mode.
   // "Apply relative position": Apply relative target position in relative positioning mode (401).
   // "START_STOP" = Start/stop with fieldbus ramp
   // "FAULT_RESET": true: Fault reset
   // "ACTIVATE_DRIVE_TRAIN_2" = true: Activate drive train 2
   // "DEACTIVATE_SW_LIMIT_SWITCH"
   // "ACTIVATE_OUPUT_STAGE_INHIBIT" = true: Activate output stage inhibit
   // "ACTIVATE_STANDBY_MODE" = true: Activate standby mode
   // "HEARTBEAT_IN": Copied to HEARTBEAT_OUT
   // "SETPOINT_SPEED": in user unit (INT) 
   // "SETPOINT_ACCELERATION":  in user unit (INT) 
   // "SETPOINT_DECELERATION":  in user unit (INT)
   // "DIGITAL_OUTPUTS": MoviSuite/Movikit../Inputs/Outputs: dig Outputs: the setting "control via fieldbus" is needed
   // "SETPOINT_APPLICATION_MODE": Operating_Mode: 10x: Jog; 30x: Ref.; 40x: Pos.; 700: Brake test 
   //     => Manual "MOVIKIT® Positioning, Velocity"
   // "TARGET_POSITION":	Target Position in user unit (DINT)
   // 
   // Outputs of the FC:
   // 
   // If the data transmission/PROFINET is disrupted, all outputs will be deleted..
   // => "COMMUNICATION_OK = false (self-confirming)
   // "READY" = true: Ready for operation.
   // "STO_INACTIVE" = true: STO inactive.
   // "OUTPUT_STAGE_ENABLED" = true: Output stage enabled.
   // "BRAKE_RELEASED" = true: Brake released.
   // "MOTOR_TURNING" = true: Motor running
   // "ACTIVE_DRIVE_REFERENCED" = true: Active drive referenced
   // "NEW_RELATIVE_POSITION_APPLIED" = true: New relative position applied
   // "IN_POSITION_SIGNAL_ACTIVE" = true: "In position" signal active
   // "FAULT" = true: Fault.
   // "WARNING" = true: Warning 
   // "DRIVE_TRAIN_2_ACTIVE" = true: Drive train 2 active.
   // "SETPOINT-ACTUAL_COMPARISON"
   // "SW_LIMIT_SWITCHES_INACTIVE" = true: Software limit switches inactive
   //  "STANDBY_MODE_INACTIVE" = true: Stand-by Mode is active.
   // "HEARTBEAT_OUT" : This signal is copied internally from "HEARTBEAT_IN"
   // "ACTUAL_SPEED": in user unit (INT) 
   // "STATUS_MAIN_FAULT_SUB_FAULT:" (WORD)
   //    No fault: Display of current FCB; fault/warning:  High-Byte Fault; Low-Byte SubFault
   // "ACTUAL_TORQUE":in user unit (INT)
   // "DIGITAL_INPUTS" : The digital inputs are read out
   // "ACTUAL_APPLICATION_MODE":	Actual Operating_Mode: 10x: Jog; 30x: Ref.; 40x: Pos.; 700: Brake test 
   //     => Manual "MOVIKIT® Positioning, Velocity"
   // "ACTUAL_POSITION":	 Actual Position in user unit (DINT)
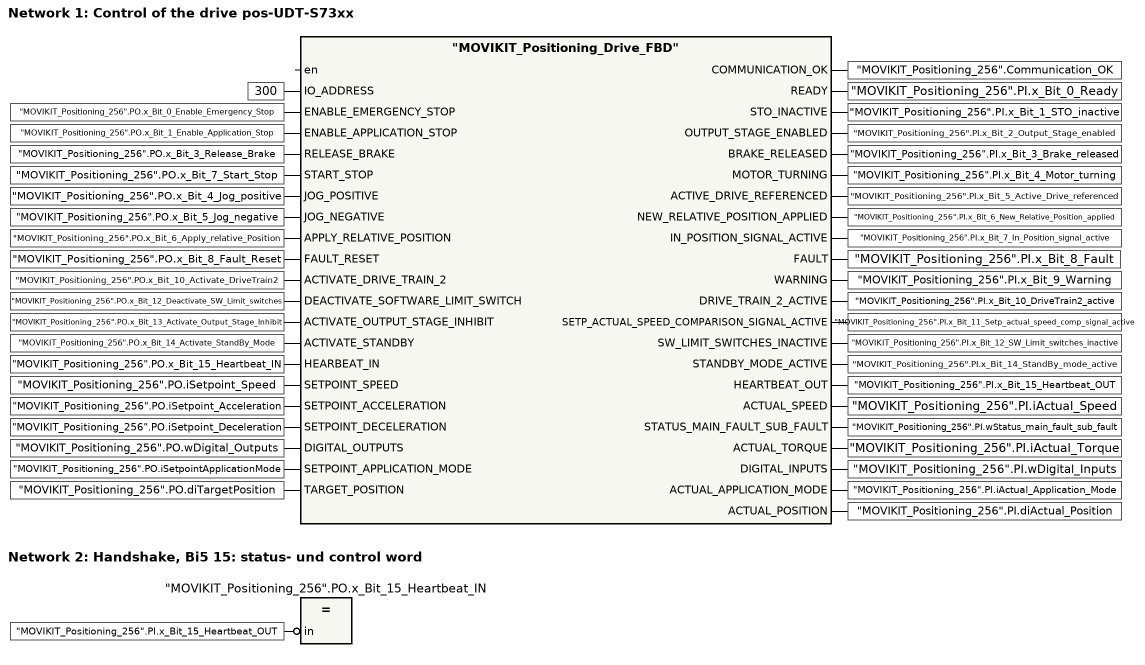
   "MOVIKIT_Positioning_Drive_FBD"(IO_ADDRESS := 300,
                           ENABLE_EMERGENCY_STOP := "MOVIKIT_Positioning_256".PO.x_Bit_0_Enable_Emergency_Stop,
                           ENABLE_APPLICATION_STOP := "MOVIKIT_Positioning_256".PO.x_Bit_1_Enable_Application_Stop,
                           RELEASE_BRAKE := "MOVIKIT_Positioning_256".PO.x_Bit_3_Release_Brake,
                           START_STOP := "MOVIKIT_Positioning_256".PO.x_Bit_7_Start_Stop,
                           JOG_POSITIVE := "MOVIKIT_Positioning_256".PO.x_Bit_4_Jog_positive,
                           JOG_NEGATIVE := "MOVIKIT_Positioning_256".PO.x_Bit_5_Jog_negative,
                           APPLY_RELATIVE_POSITION := "MOVIKIT_Positioning_256".PO.x_Bit_6_Apply_relative_Position,
                           FAULT_RESET := "MOVIKIT_Positioning_256".PO.x_Bit_8_Fault_Reset,
                           ACTIVATE_DRIVE_TRAIN_2 := "MOVIKIT_Positioning_256".PO.x_Bit_10_Activate_DriveTrain2,
                           DEACTIVATE_SOFTWARE_LIMIT_SWITCH := "MOVIKIT_Positioning_256".PO.x_Bit_12_Deactivate_SW_Limit_switches,
                           ACTIVATE_OUTPUT_STAGE_INHIBIT := "MOVIKIT_Positioning_256".PO.x_Bit_13_Activate_Output_Stage_Inhibit,
                           ACTIVATE_STANDBY := "MOVIKIT_Positioning_256".PO.x_Bit_14_Activate_StandBy_Mode,
                           HEARBEAT_IN := "MOVIKIT_Positioning_256".PO.x_Bit_15_Heartbeat_IN,
                           SETPOINT_SPEED := "MOVIKIT_Positioning_256".PO.iSetpoint_Speed,
                           SETPOINT_ACCELERATION := "MOVIKIT_Positioning_256".PO.iSetpoint_Acceleration,
                           SETPOINT_DECELERATION := "MOVIKIT_Positioning_256".PO.iSetpoint_Deceleration,
                           DIGITAL_OUTPUTS := "MOVIKIT_Positioning_256".PO.wDigital_Outputs,
                           SETPOINT_APPLICATION_MODE := "MOVIKIT_Positioning_256".PO.iSetpointApplicationMode,
                           TARGET_POSITION := "MOVIKIT_Positioning_256".PO.diTargetPosition,
                           COMMUNICATION_OK => "MOVIKIT_Positioning_256".Communication_OK,
                           READY => "MOVIKIT_Positioning_256".PI.x_Bit_0_Ready,
                           STO_INACTIVE => "MOVIKIT_Positioning_256".PI.x_Bit_1_STO_inactive,
                           OUTPUT_STAGE_ENABLED => "MOVIKIT_Positioning_256".PI.x_Bit_2_Output_Stage_enabled,
                           BRAKE_RELEASED => "MOVIKIT_Positioning_256".PI.x_Bit_3_Brake_released,
                           MOTOR_TURNING => "MOVIKIT_Positioning_256".PI.x_Bit_4_Motor_turning,
                           ACTIVE_DRIVE_REFERENCED => "MOVIKIT_Positioning_256".PI.x_Bit_5_Active_Drive_referenced,
                           NEW_RELATIVE_POSITION_APPLIED => "MOVIKIT_Positioning_256".PI.x_Bit_6_New_Relative_Position_applied,
                           IN_POSITION_SIGNAL_ACTIVE => "MOVIKIT_Positioning_256".PI.x_Bit_7_In_Position_signal_active,
                           FAULT => "MOVIKIT_Positioning_256".PI.x_Bit_8_Fault,
                           WARNING => "MOVIKIT_Positioning_256".PI.x_Bit_9_Warning,
                           DRIVE_TRAIN_2_ACTIVE => "MOVIKIT_Positioning_256".PI.x_Bit_10_DriveTrain2_active,
                           SETP_ACTUAL_SPEED_COMPARISON_SIGNAL_ACTIVE => "MOVIKIT_Positioning_256".PI.x_Bit_11_Setp_actual_speed_comp_signal_active,
                           SW_LIMIT_SWITCHES_INACTIVE => "MOVIKIT_Positioning_256".PI.x_Bit_12_SW_Limit_switches_inactive,
                           STANDBY_MODE_ACTIVE => "MOVIKIT_Positioning_256".PI.x_Bit_14_StandBy_mode_active,
                           HEARTBEAT_OUT => "MOVIKIT_Positioning_256".PI.x_Bit_15_Heartbeat_OUT,
                           ACTUAL_SPEED => "MOVIKIT_Positioning_256".PI.iActual_Speed,
                           STATUS_MAIN_FAULT_SUB_FAULT => "MOVIKIT_Positioning_256".PI.wStatus_main_fault_sub_fault,
                           ACTUAL_TORQUE => "MOVIKIT_Positioning_256".PI.iActual_Torque,
                           DIGITAL_INPUTS => "MOVIKIT_Positioning_256".PI.wDigital_Inputs,
                           ACTUAL_APPLICATION_MODE => "MOVIKIT_Positioning_256".PI.iActual_Application_Mode,
                           ACTUAL_POSITION => "MOVIKIT_Positioning_256".PI.diActual_Position);
END_REGION

REGION Network 2: Handshake, Bi5 15: status- und control word
   "MOVIKIT_Positioning_256".PO.x_Bit_15_Heartbeat_IN := NOT "MOVIKIT_Positioning_256".PI.x_Bit_15_Heartbeat_OUT;
END_REGION
END_FUNCTION

FUNCTION "MOVIKIT_Positioning_Drive_FBD" : Void   // FC142, FBD
TITLE = MOVIKIT Positioning Drive/S73xx in FBD
{ S7_Optimized_Access := 'FALSE' }
AUTHOR : CSCEASDI
FAMILY : MOVIKIT
VERSION : 2.1
// This sample program only demonstrates the basic approach. We do not accept any legal or other liability for incorrect program functions and their consequences!
// 
// The FC142 serves as a program module for controlling the MOVIKIT module "Positioning Drive" for the Generation C device series. With the help of the FC142, the converters can be controlled via PROFINET IO/PROFIBUS DP. 
// 
// Device & networks: To use this FC, a 8 PD slot must be configured.
// 
// This FC uses the UDTs "SEW_MOVIKIT_PositioningDrive_SETPOINTS_V2.1" and "SEW_MOVIKIT_PositioningDrive_STATUS_V2.1". Please make sure that these PLC data types are available in your TIA project. These UDTs can be copied from the original TIA sample project or from the MOVIKIT_Vel_&_Pos_UDTs_V2.1.al14 library.
// 
// Attention! 
// S73xx/4xx:"IO_ADDRESS"/Data Type Word:  Assign the peripheral address of the 8 PD slot;
// S71xxx: "IO_ADDRESS" change the data type from Word to "HW_IO". Assign the HW-Identifier of the 8PD slot.
   VAR_INPUT
      IO_ADDRESS : Word;   // S73xx/4xx:"IO_ADDRESS"/Data Type Word: Assign the peripheral address of the 5 PD slot; S71xxx: "IO_ADDRESS" change the data type from Word to "HW_IO". Assign the HW-Identifier of the 5 PD slot.
      ENABLE_EMERGENCY_STOP : Bool;   // true: Enable; false: emergency stop
      ENABLE_APPLICATION_STOP : Bool;   // true: Enable; false: Application stop
      RELEASE_BRAKE : Bool;   // true: release brake (without enable)
      START_STOP : Bool;   // Start/stop with fieldbus ramp
      JOG_POSITIVE : Bool;   // true: Jog positive
      JOG_NEGATIVE : Bool;   // true: Jog negative
      APPLY_RELATIVE_POSITION : Bool;   // true: Apply relative position
      FAULT_RESET : Bool;   // true: Fault reset
      ACTIVATE_DRIVE_TRAIN_2 : Bool;   // true: Activate drive train 2
      DEACTIVATE_SOFTWARE_LIMIT_SWITCH : Bool;   // true: Deactivate software limit switches
      ACTIVATE_OUTPUT_STAGE_INHIBIT : Bool;   // true: Activate output stage inhibit
      ACTIVATE_STANDBY : Bool;   // true: Activate standby mode
      HEARBEAT_IN : Bool;   // Copied to HEARTBEAT_OUT
      SETPOINT_SPEED : Int;   // in user unit (INT)
      SETPOINT_ACCELERATION : Int;   // in user unit (INT)
      SETPOINT_DECELERATION : Int;   // in user unit (INT)
      DIGITAL_OUTPUTS : Word;   // MoviSuite/Movikit../Inputs/Outputs: dig Outputs: the setting "control via fieldbus" is needed
      SETPOINT_APPLICATION_MODE : Int;   // Operating_Mode: 10x: Jog; 30x: Ref.; 40x: Pos.; 700: Brake test => Manual "MOVIKIT® Positioning, Velocity"
      TARGET_POSITION : DInt;   // Target Position in user unit
   END_VAR
   VAR_OUTPUT
      COMMUNICATION_OK : Bool;   // true: DPRD_DAT and DPWR_DAT are working correctly. false: 5 PD slot required; Check address at Input "IO_ADDRESS"
      READY : Bool;   // true: Ready for operation.
      STO_INACTIVE : Bool;   // true: STO inactive.
      OUTPUT_STAGE_ENABLED : Bool;   // true: Output stage enabled.
      BRAKE_RELEASED : Bool;   // true: Brake released.
      MOTOR_TURNING : Bool;   // true: Motor turning.
      ACTIVE_DRIVE_REFERENCED : Bool;   // true: Active drive referenced
      NEW_RELATIVE_POSITION_APPLIED : Bool;   // true: New relative position applied
      IN_POSITION_SIGNAL_ACTIVE : Bool;   // true: "In position" signal active
      FAULT : Bool;   // true: Fault.
      WARNING : Bool;   // true: Warning
      DRIVE_TRAIN_2_ACTIVE : Bool;   // true: Drive train 2 active.
      SETP_ACTUAL_SPEED_COMPARISON_SIGNAL_ACTIVE : Bool;
      SW_LIMIT_SWITCHES_INACTIVE : Bool;   // true: Software limit switches inactive
      STANDBY_MODE_ACTIVE : Bool;   // true: Stand-by Mode is active.
      HEARTBEAT_OUT : Bool;   // This signal is copied internally from "HEARTBEAT_IN"
      ACTUAL_SPEED : Int;   // in user unit (INT)
      STATUS_MAIN_FAULT_SUB_FAULT : Word;   // No fault: Display of current FCB; fault/warning: High-Byte Fault; Low-Byte SubFault
      ACTUAL_TORQUE : Int;   // in user unit (INT)
      DIGITAL_INPUTS : Word;   // The digital inputs are read out
      ACTUAL_APPLICATION_MODE : Int;   // Actual Operating_Mode: 10x: Jog; 30x: Ref.; 40x: Pos.; 700: Brake test => Manual "MOVIKIT® Positioning, Velocity"
      ACTUAL_POSITION : DInt;   // Actual Position in user unit
   END_VAR
   VAR_TEMP
      PI : "SEW_MOVIKIT_PositioningDrive_STATUS_V2.1";
      PO : "SEW_MOVIKIT_PositioningDrive_SETPOINTS_V2.1";
      DPRD_RET_VAL : Int;
      DPWR_RET_VAL : Int;
      FALSE : Bool;
   END_VAR
   VAR_TEMP   // added for the SCL form of the ladder/FBD networks
      _w1 : Bool;
   END_VAR
BEGIN

REGION Network 1: Def."#FALSE"
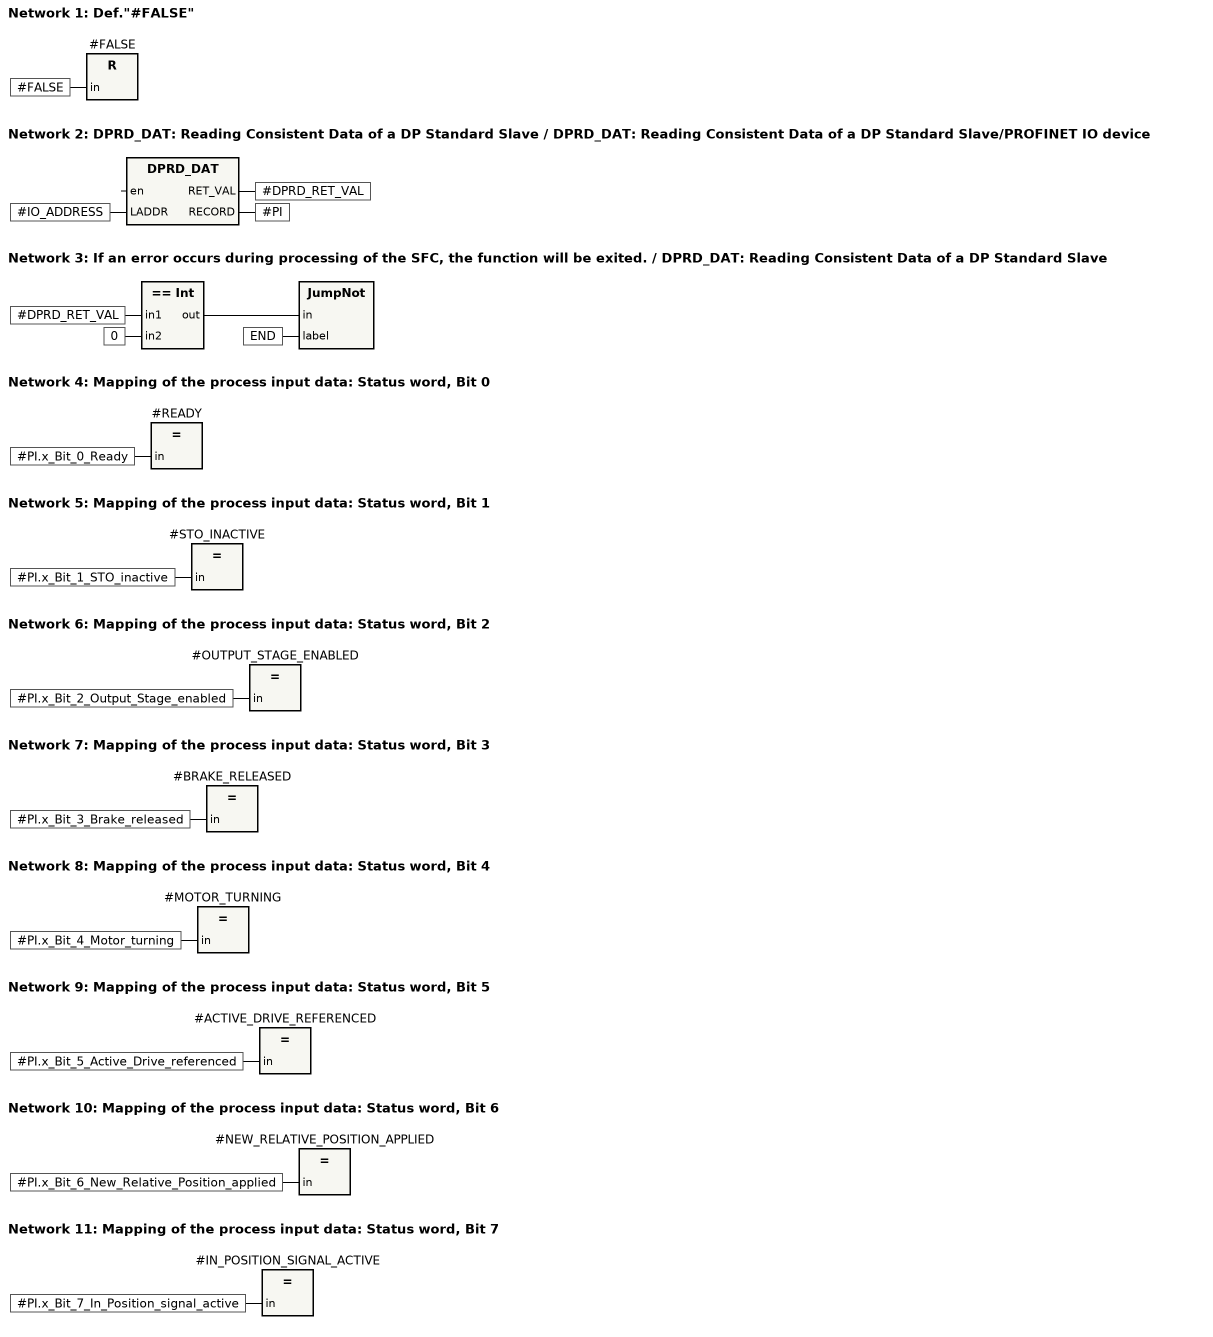
   IF #FALSE THEN #FALSE := FALSE; END_IF;
END_REGION

REGION Network 2: DPRD_DAT: Reading Consistent Data of a DP Standard Slave / DPRD_DAT: Reading Consistent Data of a DP Standard Slave/PROFINET IO device
   #DPRD_RET_VAL := DPRD_DAT(LADDR := #IO_ADDRESS, RECORD => #PI);
END_REGION

REGION Network 3: If an error occurs during processing of the SFC, the function will be exited. / DPRD_DAT: Reading Consistent Data of a DP Standard Slave
   // If the return value = 0, COM_DPRD_OK = TRUE. The function is further processed and not jumped to "END".
   // no SCL statement known for JumpNot: written as a call
   JumpNot(in := #DPRD_RET_VAL = 0, label := END);
END_REGION

REGION Network 4: Mapping of the process input data: Status word, Bit 0
   #READY := #PI.x_Bit_0_Ready;
END_REGION

REGION Network 5: Mapping of the process input data: Status word, Bit 1
   #STO_INACTIVE := #PI.x_Bit_1_STO_inactive;
END_REGION

REGION Network 6: Mapping of the process input data: Status word, Bit 2
   #OUTPUT_STAGE_ENABLED := #PI.x_Bit_2_Output_Stage_enabled;
END_REGION

REGION Network 7: Mapping of the process input data: Status word, Bit 3
   #BRAKE_RELEASED := #PI.x_Bit_3_Brake_released;
END_REGION

REGION Network 8: Mapping of the process input data: Status word, Bit 4
   #MOTOR_TURNING := #PI.x_Bit_4_Motor_turning;
END_REGION

REGION Network 9: Mapping of the process input data: Status word, Bit 5
   #ACTIVE_DRIVE_REFERENCED := #PI.x_Bit_5_Active_Drive_referenced;
END_REGION

REGION Network 10: Mapping of the process input data: Status word, Bit 6
   #NEW_RELATIVE_POSITION_APPLIED := #PI.x_Bit_6_New_Relative_Position_applied;
END_REGION

REGION Network 11: Mapping of the process input data: Status word, Bit 7
   #IN_POSITION_SIGNAL_ACTIVE := #PI.x_Bit_7_In_Position_signal_active;
END_REGION

REGION Network 12: Mapping of the process input data: Status word, Bit 8
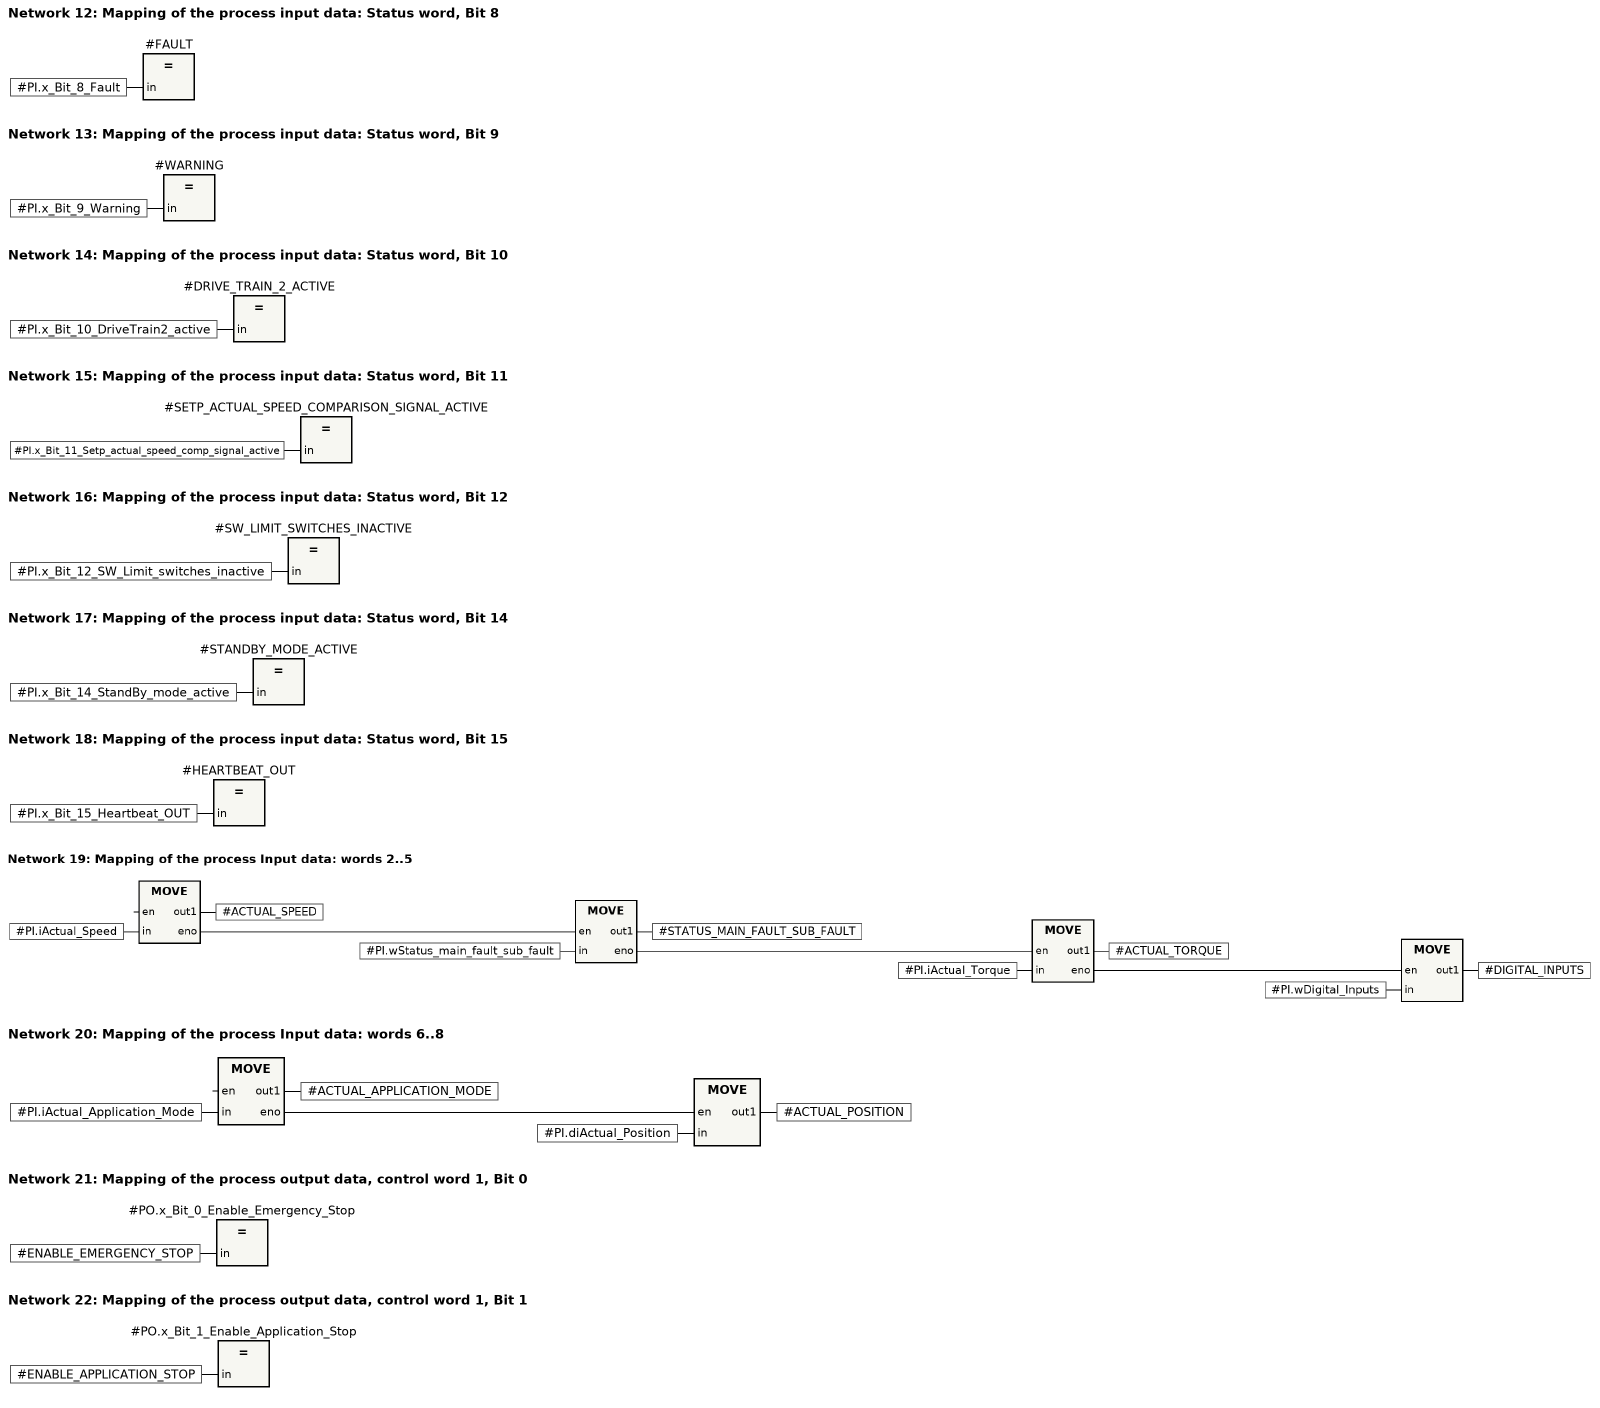
   #FAULT := #PI.x_Bit_8_Fault;
END_REGION

REGION Network 13: Mapping of the process input data: Status word, Bit 9
   #WARNING := #PI.x_Bit_9_Warning;
END_REGION

REGION Network 14: Mapping of the process input data: Status word, Bit 10
   #DRIVE_TRAIN_2_ACTIVE := #PI.x_Bit_10_DriveTrain2_active;
END_REGION

REGION Network 15: Mapping of the process input data: Status word, Bit 11
   #SETP_ACTUAL_SPEED_COMPARISON_SIGNAL_ACTIVE := #PI.x_Bit_11_Setp_actual_speed_comp_signal_active;
END_REGION

REGION Network 16: Mapping of the process input data: Status word, Bit 12
   #SW_LIMIT_SWITCHES_INACTIVE := #PI.x_Bit_12_SW_Limit_switches_inactive;
END_REGION

REGION Network 17: Mapping of the process input data: Status word, Bit 14
   #STANDBY_MODE_ACTIVE := #PI.x_Bit_14_StandBy_mode_active;
END_REGION

REGION Network 18: Mapping of the process input data: Status word, Bit 15
   #HEARTBEAT_OUT := #PI.x_Bit_15_Heartbeat_OUT;
END_REGION

REGION Network 19: Mapping of the process Input data: words 2..5
   // ENO of a box is taken as its EN; it also drops when the box reports an error
   #ACTUAL_SPEED := #PI.iActual_Speed;
   #STATUS_MAIN_FAULT_SUB_FAULT := #PI.wStatus_main_fault_sub_fault;
   #ACTUAL_TORQUE := #PI.iActual_Torque;
   #DIGITAL_INPUTS := #PI.wDigital_Inputs;
END_REGION

REGION Network 20: Mapping of the process Input data: words 6..8
   // ENO of a box is taken as its EN; it also drops when the box reports an error
   #ACTUAL_APPLICATION_MODE := #PI.iActual_Application_Mode;
   #ACTUAL_POSITION := #PI.diActual_Position;
END_REGION

REGION Network 21: Mapping of the process output data, control word 1, Bit 0
   #PO.x_Bit_0_Enable_Emergency_Stop := #ENABLE_EMERGENCY_STOP;
END_REGION

REGION Network 22: Mapping of the process output data, control word 1, Bit 1
   #PO.x_Bit_1_Enable_Application_Stop := #ENABLE_APPLICATION_STOP;
END_REGION

REGION Network 23: Mapping of the process output data, control word 1, Bit 3
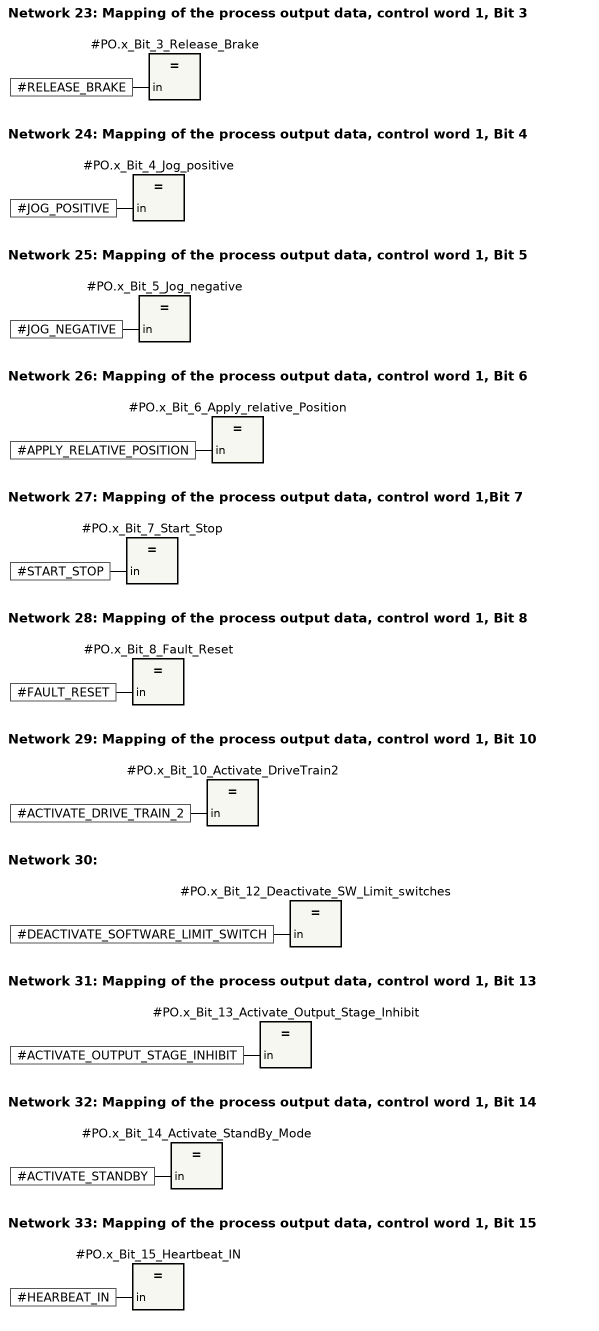
   #PO.x_Bit_3_Release_Brake := #RELEASE_BRAKE;
END_REGION

REGION Network 24: Mapping of the process output data, control word 1, Bit 4
   #PO.x_Bit_4_Jog_positive := #JOG_POSITIVE;
END_REGION

REGION Network 25: Mapping of the process output data, control word 1, Bit 5
   #PO.x_Bit_5_Jog_negative := #JOG_NEGATIVE;
END_REGION

REGION Network 26: Mapping of the process output data, control word 1, Bit 6
   #PO.x_Bit_6_Apply_relative_Position := #APPLY_RELATIVE_POSITION;
END_REGION

REGION Network 27: Mapping of the process output data, control word 1,Bit 7
   #PO.x_Bit_7_Start_Stop := #START_STOP;
END_REGION

REGION Network 28: Mapping of the process output data, control word 1, Bit 8
   #PO.x_Bit_8_Fault_Reset := #FAULT_RESET;
END_REGION

REGION Network 29: Mapping of the process output data, control word 1, Bit 10
   #PO.x_Bit_10_Activate_DriveTrain2 := #ACTIVATE_DRIVE_TRAIN_2;
END_REGION

REGION Network 30
   #PO.x_Bit_12_Deactivate_SW_Limit_switches := #DEACTIVATE_SOFTWARE_LIMIT_SWITCH;
END_REGION

